	MEMSET(ADR(stMetsEfficiency.PackProduced), 16#00, SIZEOF(stMetsEfficiency.PackProduced));
	MEMSET(ADR(stMetsEfficiency.OutersProduced), 16#00, SIZEOF(stMetsEfficiency.OutersProduced));
	MEMSET(ADR(stMetsEfficiency.CaseProduced), 16#00, SIZEOF(stMetsEfficiency.CaseProduced));

	stMetsEfficiency.MachineID.ProductionSite	 := sProductionSite;
	stMetsEfficiency.MachineID.ProductionLine	:= sPCM;
	stMetsEfficiency.StartDateTime 			:= F_SYSTEM_SystemTimeAsISO8601(stCTDateTime.sSystemTime, stCTDateTime.sUTCTimeZoneOffset );
	stMetsEfficiency.CodingAndTrackingMode 	:= stPCMStatus.nOpMode;
	stMetsEfficiency.AcceptanceLevel  			:= stPCMStatus.nAcceptanceLevel;
	stMetsEfficiency.PacksPerOuter			:= stPCMStatus.nPacksPerOuter;

	MEMSET(ADR(stBarGraph), 16#00, SIZEOF(stBarGraph));

	bTimerFlag:=TRUE;
END_IF

tofDoneTimer(IN:=bTimerFlag,PT:=t#5s, Q=>bDone);

END_FUNCTION_BLOCK

// ---- POUs/METS/Common LIB/06_KPI LIB/ClearStatistic/FB_KPI_ClearGeneraStatistic.TcPOU
FUNCTION_BLOCK FB_KPI_ClearGeneraStatistic
VAR_INPUT
	bExecute				: BOOL;
	stCTDateTime			: ST_SYSTEM_DateTime;	(* CaseTrace date/time structure *)
	sProductionSite		: STRING(4);
	sPCM				: STRING(4);
	bForceNovReset		: BOOL;
END_VAR
VAR_IN_OUT

	stPCMStatus			: ST_PCM_Status;

	stMetsCameras			: ST_NOVRAM_METS_Cameras;
	stMetsEfficiency		: ST_NOVRAM_METS_Inspection;
	stCasePackerSignals		: ST_NOVRAM_METS_DualInputs;
	stCaseInspactionLog		: ST_NOVRAM_METS_CaseInspactionLog;
	
	stShiftStatistic		: ST_NOVRAM_METS_EventCounters; 
	stProdStatistic			: ST_NOVRAM_METS_EventCounters; 

	stBarGraph			: ST_HMI_BarGraph;

	stWriteOACFileStatistic		: ST_FILE_WriteFileStatistic;	(*Move to METSEfficency one day*)
	stWriteCHMFileStatistic		: ST_FILE_WriteFileStatistic;	(*Move to METSEfficency one day*)

END_VAR
VAR_OUTPUT
	bDone				: BOOL;
END_VAR
VAR
	fbExecute 			: R_TRIG;
	bTimerFlag			: BOOL;
	tofDoneTimer			: TOF;

	nCounter				: INT;


END_VAR

(* rising edge of bExecute *)
fbExecute(CLK:= bExecute);

bTimerFlag:=FALSE;

IF fbExecute.Q THEN

	nCounter := nCounter +1;

	MEMSET(ADR(stMetsCameras), 16#00, SIZEOF(stMetsCameras));
	MEMSET(ADR(stMetsEfficiency), 16#00, SIZEOF(stMetsEfficiency));
	MEMSET(ADR(stCasePackerSignals), 16#00, SIZEOF(stCasePackerSignals));
	MEMSET(ADR(stCaseInspactionLog), 16#00, SIZEOF(stCaseInspactionLog));

	stMetsCameras.MachineID.ProductionSite 	:= sProductionSite;
	stMetsCameras.MachineID.ProductionLine	:= sPCM;
	stMetsCameras.StartDateTime 				:=  F_SYSTEM_SystemTimeAsISO8601(stCTDateTime.sSystemTime, stCTDateTime.sUTCTimeZoneOffset );
	stMetsCameras.CodingAndTrackingMode 	:= stPCMStatus.nOpMode;

	stMetsEfficiency.MachineID.ProductionSite	 := sProductionSite;
	stMetsEfficiency.MachineID.ProductionLine	:= sPCM;
	stMetsEfficiency.StartDateTime 			:= F_SYSTEM_SystemTimeAsISO8601(stCTDateTime.sSystemTime, stCTDateTime.sUTCTimeZoneOffset );
	stMetsEfficiency.CodingAndTrackingMode 	:= stPCMStatus.nOpMode;
	stMetsEfficiency.AcceptanceLevel  			:= stPCMStatus.nAcceptanceLevel;
	stMetsEfficiency.PacksPerOuter			:= stPCMStatus.nPacksPerOuter;

	stCasePackerSignals.MachineID.ProductionSite	 := sProductionSite;
	stCasePackerSignals.MachineID.ProductionLine	:= sPCM;
	stCasePackerSignals.StartDateTime 				:=  F_SYSTEM_SystemTimeAsISO8601(stCTDateTime.sSystemTime, stCTDateTime.sUTCTimeZoneOffset );
	stCasePackerSignals.CodingAndTrackingMode	 	:=stPCMStatus.nOpMode;

	stCaseInspactionLog.MachineID.ProductionSite 	:= sProductionSite;
	stCaseInspactionLog.MachineID.ProductionLine	:= sPCM;
	stCaseInspactionLog.StartDateTime 				:=  F_SYSTEM_SystemTimeAsISO8601(stCTDateTime.sSystemTime, stCTDateTime.sUTCTimeZoneOffset );
	stCaseInspactionLog.CodingAndTrackingMode		:= stPCMStatus.nOpMode;
	stCaseInspactionLog.nPacksPerCase  			:= stPCMStatus.nPacksPerCase;
	stCaseInspactionLog.nOutersPerCase			:= stPCMStatus.nOutersPerCase;

	MEMSET(ADR(stBarGraph), 16#00, SIZEOF(stBarGraph));

	MEMSET(ADR(stWriteOACFileStatistic), 16#00, SIZEOF(stWriteOACFileStatistic));
	MEMSET(ADR(stWriteCHMFileStatistic), 16#00, SIZEOF(stWriteCHMFileStatistic));

	bTimerFlag:=TRUE;
END_IF

tofDoneTimer(IN:=bTimerFlag,PT:=t#5s, Q=>bDone);

IF bForceNovReset THEN
	MEMSET(ADR(stShiftStatistic), 16#00, SIZEOF(stShiftStatistic));
	MEMSET(ADR(stProdStatistic), 16#00, SIZEOF(stProdStatistic));
END_IF

END_FUNCTION_BLOCK

// ---- POUs/METS/Common LIB/06_KPI LIB/ClearStatistic/FB_KPI_ClearInspectionStatistic.TcPOU
FUNCTION_BLOCK FB_KPI_ClearInspectionStatistic
VAR_INPUT
	bExecute						: BOOL;
	stCTDateTime					: ST_SYSTEM_DateTime;	(* CaseTrace date/time structure *)
	nLowerCameraGroupIndex		: INT;
	nUpperCameraGroupIndex		: INT;
END_VAR
VAR_IN_OUT
	stEfficiencyToBeCleared			: ST_KPI_InspectionEfficency;
	stMetsCameras					: ST_NOVRAM_METS_Cameras;
END_VAR
VAR_OUTPUT
	bDone				: BOOL;
END_VAR
VAR
	fbExecute 			: R_TRIG;
	bTimerFlag			: BOOL;
	tofDoneTimer			: TOF;
	nIndex				: INT;

	nCounter				: INT;
END_VAR

(* rising edge of bExecute *)
fbExecute(CLK:= bExecute);

bTimerFlag:=FALSE;

IF fbExecute.Q THEN

	nCounter := nCounter +1;



	MEMSET(ADR(stEfficiencyToBeCleared), 16#00, SIZEOF(stEfficiencyToBeCleared));

	(*stEfficiencyToBeCleared.StartDateTime 			:= F_SYSTEM_SystemTimeAsISO8601(stCTDateTime.sSystemTime, stCTDateTime.sUTCTimeZoneOffset );*)

	IF nLowerCameraGroupIndex > 0 	AND
		nLowerCameraGroupIndex <= nUpperCameraGroupIndex THEN

		FOR nIndex :=nLowerCameraGroupIndex  TO MIN(nUpperCameraGroupIndex, cMAX_CAMERA_NUMBER)  DO
			MEMSET(ADR(stMetsCameras.aCameraEvaluation[nIndex]), 16#00, SIZEOF(stMetsCameras.aCameraEvaluation[nIndex]));
		END_FOR
	END_IF

	bTimerFlag:=TRUE;
END_IF

tofDoneTimer(IN:=bTimerFlag,PT:=t#5s, Q=>bDone);

END_FUNCTION_BLOCK

// ---- POUs/METS/Common LIB/06_KPI LIB/ClearStatistic/FB_KPI_ClearPackOuterInspection.TcPOU
FUNCTION_BLOCK FB_KPI_ClearPackOuterInspection
VAR_INPUT
	bExecute						: BOOL;
	stCTDateTime					: ST_SYSTEM_DateTime;	(* CaseTrace date/time structure *)
	sProductionSite				: STRING(4);
	sPCM						: STRING(4);
END_VAR
VAR_IN_OUT

	stPCMStatus					: ST_PCM_Status;
	stMetsEfficiency		: ST_NOVRAM_METS_Inspection;

END_VAR
VAR_OUTPUT
	bDone				: BOOL;
END_VAR
VAR
	fbExecute 			: R_TRIG;
	bTimerFlag			: BOOL;
	tofDoneTimer			: TOF;

	nCounter				: INT;
END_VAR

(* rising edge of bExecute *)
fbExecute(CLK:= bExecute);

bTimerFlag:=FALSE;

IF fbExecute.Q THEN

	nCounter := nCounter +1;

	stMetsEfficiency.MachineID.ProductionSite	 := sProductionSite;
	stMetsEfficiency.MachineID.ProductionLine	:= sPCM;
	stMetsEfficiency.StartDateTime 			:= F_SYSTEM_SystemTimeAsISO8601(stCTDateTime.sSystemTime, stCTDateTime.sUTCTimeZoneOffset );
	stMetsEfficiency.CodingAndTrackingMode 	:= stPCMStatus.nOpMode;
	stMetsEfficiency.AcceptanceLevel  			:= stPCMStatus.nAcceptanceLevel;
	stMetsEfficiency.PacksPerOuter			:= stPCMStatus.nPacksPerOuter;

	MEMSET(ADR(stMetsEfficiency.OutersProcessing), 16#00, SIZEOF(stMetsEfficiency.OutersProcessing));
	MEMSET(ADR(stMetsEfficiency.OCVFileEfficiency), 16#00, SIZEOF(stMetsEfficiency.OCVFileEfficiency));
	MEMSET(ADR(stMetsEfficiency.PacksRead), 16#00, SIZEOF(stMetsEfficiency.PacksRead));
	MEMSET(ADR(stMetsEfficiency.PackPosEfficiency), 16#00, SIZEOF(stMetsEfficiency.PackPosEfficiency));

	MEMSET(ADR(stMetsEfficiency.PackAggregationEfficiency), 16#00, SIZEOF(stMetsEfficiency.PackAggregationEfficiency));

	MEMSET(ADR(stMetsEfficiency.aConfirmCodeEfficiency), 16#00, SIZEOF(stMetsEfficiency.aConfirmCodeEfficiency));
	MEMSET(ADR(stMetsEfficiency.PackConfirmationEfficiency), 16#00, SIZEOF(stMetsEfficiency.PackConfirmationEfficiency));
	MEMSET(ADR(stMetsEfficiency.OuterValidationEfficiency), 16#00, SIZEOF(stMetsEfficiency.OuterValidationEfficiency));
	MEMSET(ADR(stMetsEfficiency.OuterAggregationEfficiency), 16#00, SIZEOF(stMetsEfficiency.OuterAggregationEfficiency));

	bTimerFlag:=TRUE;
END_IF

tofDoneTimer(IN:=bTimerFlag,PT:=t#5s, Q=>bDone);

END_FUNCTION_BLOCK

// ---- POUs/METS/Common LIB/06_KPI LIB/ItemEfficiency/FB_KPI_CaseEfficiency.TcPOU
FUNCTION_BLOCK FB_KPI_CaseEfficiency
VAR_INPUT
	bUpdateItemData		: 	BOOL;
	bItemSuccessful		:	 BOOL;
END_VAR
VAR_IN_OUT
	stItemInspection		: 	ST_KPI_InspectionEfficency;
END_VAR
VAR_OUTPUT
END_VAR
VAR
	rtrigUpdateItemData	:	 R_TRIG;
END_VAR

rtrigUpdateItemData(CLK:= bUpdateItemData);

IF rtrigUpdateItemData.Q THEN

	stItemInspection.ProcessedTotal :=  stItemInspection.ProcessedTotal + 1;
		IF bItemSuccessful THEN
			stItemInspection.ProcessedSuccessful := stItemInspection.ProcessedSuccessful + 1;
		ELSE
			stItemInspection.ProcessedRejected := stItemInspection.ProcessedRejected + 1;
		END_IF
END_IF

stItemInspection.ProcessedEfficiency := F_SafeDIV(stItemInspection.ProcessedSuccessful  * 100,  stItemInspection.ProcessedTotal);
stItemInspection.ProcessedEfficiency :=LIMIT(0, stItemInspection.ProcessedEfficiency, 100);

END_FUNCTION_BLOCK

// ---- POUs/METS/Common LIB/06_KPI LIB/ItemEfficiency/FB_KPI_InterimEfficiency.TcPOU
FUNCTION_BLOCK FB_KPI_InterimEfficiency
VAR_INPUT
	bUpdateItemData		: 	BOOL;
	bItemSuccessful		:	 BOOL;
END_VAR
VAR_IN_OUT
	stItemInspection		: 	ST_KPI_InspectionEfficency;
END_VAR
VAR_OUTPUT
END_VAR
VAR
	rtrigUpdateItemData	:	 R_TRIG;
END_VAR

rtrigUpdateItemData(CLK:= bUpdateItemData);

IF rtrigUpdateItemData.Q THEN

	stItemInspection.ProcessedTotal :=  stItemInspection.ProcessedTotal + 1;
		IF bItemSuccessful THEN
			stItemInspection.ProcessedSuccessful := stItemInspection.ProcessedSuccessful + 1;
		ELSE
			stItemInspection.ProcessedRejected := stItemInspection.ProcessedRejected + 1;
		END_IF
END_IF

stItemInspection.ProcessedEfficiency := F_SafeDIV(stItemInspection.ProcessedSuccessful  * 100,  stItemInspection.ProcessedTotal);
stItemInspection.ProcessedEfficiency :=LIMIT(0, stItemInspection.ProcessedEfficiency, 100);

END_FUNCTION_BLOCK

// ---- POUs/METS/Common LIB/06_KPI LIB/ItemEfficiency/FB_KPI_OutersEfficiency.TcPOU
FUNCTION_BLOCK FB_KPI_OutersEfficiency
VAR_INPUT
	ePackAggregationMode			: E_SYSTEM_PackAggregationMode ;
	bUpdateAtConfimrationCamera	: BOOL;
	bUpdateAtValidationCamera		: BOOL;
	bUpdateTotal						: BOOL;
	bUpdateConfirmCam				: BOOL;
	bUpdateValidCam					: BOOL;

	bItemSuccessful					: BOOL;

	nPackEntireLength					: INT;
	nOuterEntireLength				: INT;
	nValidCamExpectedResp			: INT;

END_VAR
VAR_IN_OUT
	stConfirmationCameraImage		: ST_SCANNER_ImageData;		(* image data structure *)
	stValidationCameraImage			: ST_SCANNER_ImageData;		(* image data structure *)

	stMetsEfficiency					: ST_NOVRAM_METS_Inspection;
END_VAR
VAR_OUTPUT
END_VAR
VAR
	rtrigUpdateAtConfimrationCamera	: R_TRIG;
	rtrigUpdateAtValidationCamera	: R_TRIG;
	rtrigUpdateTotal				: R_TRIG;
	rtrigUpdateConfirmCamera		: R_TRIG;
	rtrigUpdateValidCamera			: R_TRIG;
	rtrigUpdateKPI					: R_TRIG;

	nCodeLoopPerPos				: INT;

END_VAR

CASE ePackAggregationMode OF

	E_SYSTEM_PAOL_2CAM:

		SFLX();

	E_SYSTEM_PAOL_3CAM:

		PAOL();

	E_SYSTEM_PLAS_T01, E_SYSTEM_PLAS_T02, E_SYSTEM_PLAS_T03, E_SYSTEM_PLAS_T04:

		PLAS();

END_CASE

ACTION NCW:
rtrigUpdateTotal(CLK:= bUpdateTotal);

IF rtrigUpdateTotal.Q THEN

	stMetsEfficiency.OuterAggregationEfficiency.ProcessedTotal :=  stMetsEfficiency.OuterAggregationEfficiency.ProcessedTotal + 1;
		IF bItemSuccessful THEN
			stMetsEfficiency.OuterAggregationEfficiency.ProcessedSuccessful := stMetsEfficiency.OuterAggregationEfficiency.ProcessedSuccessful + 1;
		ELSE
			stMetsEfficiency.OuterAggregationEfficiency.ProcessedRejected := stMetsEfficiency.OuterAggregationEfficiency.ProcessedRejected + 1;
		END_IF
END_IF

stMetsEfficiency.OuterAggregationEfficiency.ProcessedEfficiency :=  F_SafeDIV( UDINT_TO_LREAL(stMetsEfficiency.OuterAggregationEfficiency.ProcessedSuccessful),
																	UDINT_TO_LREAL(stMetsEfficiency.OuterAggregationEfficiency.ProcessedTotal))* 100.0;
stMetsEfficiency.OuterAggregationEfficiency.ProcessedEfficiency	:= LIMIT(0,stMetsEfficiency.OuterAggregationEfficiency.ProcessedEfficiency , 100);
END_ACTION

ACTION PAOL:
rtrigUpdateAtConfimrationCamera(CLK:= bUpdateAtConfimrationCamera);
rtrigUpdateAtValidationCamera(CLK:=bUpdateAtValidationCamera);
rtrigUpdateTotal(CLK:= bUpdateTotal);
rtrigUpdateConfirmCamera(CLK:=bUpdateConfirmCam);
rtrigUpdateValidCamera(CLK:=bUpdateValidCam);

IF rtrigUpdateAtConfimrationCamera.Q THEN
	stMetsEfficiency.OutersProcessing.AtConfimrationCamera := stMetsEfficiency.OutersProcessing.AtConfimrationCamera + 1;
END_IF

IF rtrigUpdateAtValidationCamera.Q THEN
	stMetsEfficiency.OutersProcessing.AtValidationCamera := stMetsEfficiency.OutersProcessing.AtValidationCamera + 1;
END_IF

IF rtrigUpdateTotal.Q THEN

	stMetsEfficiency.OuterAggregationEfficiency.ProcessedTotal :=stMetsEfficiency. OuterAggregationEfficiency.ProcessedTotal +1;

		IF bItemSuccessful THEN
			stMetsEfficiency.OuterAggregationEfficiency.ProcessedSuccessful := stMetsEfficiency.OuterAggregationEfficiency.ProcessedSuccessful +1;
		ELSE
			stMetsEfficiency.OuterAggregationEfficiency.ProcessedRejected  := stMetsEfficiency.OuterAggregationEfficiency.ProcessedRejected +1;
		END_IF

	stMetsEfficiency.OuterAggregationEfficiency.ProcessedEfficiency :=  F_SafeDIV( UDINT_TO_LREAL(stMetsEfficiency.OuterAggregationEfficiency.ProcessedSuccessful),
																		UDINT_TO_LREAL(stMetsEfficiency.OuterAggregationEfficiency.ProcessedTotal))* 100.0;
	stMetsEfficiency.OuterAggregationEfficiency.ProcessedEfficiency	:= LIMIT(0,stMetsEfficiency.OuterAggregationEfficiency.ProcessedEfficiency , 100);
END_IF

(************************* Update Pack Confirmation Process Efficiency*******************************************************************************)

IF rtrigUpdateConfirmCamera.Q  THEN

	stMetsEfficiency.PackConfirmationEfficiency.ProcessedTotal	:= 	stMetsEfficiency.PackConfirmationEfficiency.ProcessedTotal +1;

	IF F_PACK_ValidateCodeASCII(stConfirmationCameraImage.aCodeData[1].strDataString) =  nPackEntireLength			OR
			F_PACK_ValidateCodeASCII(stConfirmationCameraImage.aCodeData[2].strDataString) =  nPackEntireLength 	THEN

		stMetsEfficiency.PackConfirmationEfficiency.ProcessedSuccessful :=  stMetsEfficiency.PackConfirmationEfficiency.ProcessedSuccessful +1;
	ELSE
		stMetsEfficiency.PackConfirmationEfficiency.ProcessedRejected :=  stMetsEfficiency.PackConfirmationEfficiency.ProcessedRejected +1;
	END_IF

(*Confirmation Cameras Individual per pack*)
	FOR nCodeLoopPerPos := 1 TO 2 DO
		CASE LREAL_TO_INT(stConfirmationCameraImage.aCodeData[nCodeLoopPerPos].nProgramNo) OF
			1:
				IF F_PACK_ValidateCodeASCII(stConfirmationCameraImage.aCodeData[nCodeLoopPerPos].strDataString) =  nPackEntireLength THEN
					stMetsEfficiency.aConfirmCodeEfficiency[1].ReadOK :=  stMetsEfficiency.aConfirmCodeEfficiency[1].ReadOK +1;
				END_IF
			2:
				IF F_PACK_ValidateCodeASCII(stConfirmationCameraImage.aCodeData[nCodeLoopPerPos].strDataString) =  nPackEntireLength THEN
					stMetsEfficiency.aConfirmCodeEfficiency[2].ReadOK := stMetsEfficiency. aConfirmCodeEfficiency[2].ReadOK +1;
				END_IF
		END_CASE
	END_FOR

	stMetsEfficiency.PackConfirmationEfficiency.ProcessedEfficiency :=  F_SafeDIV( UDINT_TO_LREAL(stMetsEfficiency.PackConfirmationEfficiency.ProcessedSuccessful),
																	UDINT_TO_LREAL(stMetsEfficiency.PackConfirmationEfficiency.ProcessedTotal))* 100.0;
	stMetsEfficiency.PackConfirmationEfficiency.ProcessedEfficiency	:= LIMIT(0,stMetsEfficiency.PackConfirmationEfficiency.ProcessedEfficiency, 100);

	stMetsEfficiency.aConfirmCodeEfficiency[1].Efficiency :=  F_SafeDIV( UDINT_TO_LREAL(stMetsEfficiency.aConfirmCodeEfficiency[1].ReadOK),
																	UDINT_TO_LREAL(stMetsEfficiency.PackConfirmationEfficiency.ProcessedTotal))* 100.0;
	stMetsEfficiency.aConfirmCodeEfficiency[1].Efficiency	:= LIMIT(0,stMetsEfficiency.aConfirmCodeEfficiency[1].Efficiency, 100);

	stMetsEfficiency.aConfirmCodeEfficiency[2].Efficiency :=  F_SafeDIV( UDINT_TO_LREAL(stMetsEfficiency.aConfirmCodeEfficiency[2].ReadOK),
																	UDINT_TO_LREAL(stMetsEfficiency.PackConfirmationEfficiency.ProcessedTotal))* 100.0;
	stMetsEfficiency.aConfirmCodeEfficiency[2].Efficiency	:= LIMIT(0,stMetsEfficiency.aConfirmCodeEfficiency[2].Efficiency , 100);

END_IF

(************************* Update Outer Validation Process Efficiency*******************************************************************************)

IF rtrigUpdateValidCamera.Q  THEN

	stMetsEfficiency.OuterValidationEfficiency.ProcessedTotal :=	stMetsEfficiency.OuterValidationEfficiency.ProcessedTotal + 1;

	IF LEN(stValidationCameraImage.aCodeData[1].strDataString) =  nOuterEntireLength 				OR
		LEN(stValidationCameraImage.aCodeData[2].strDataString) =  nOuterEntireLength 				THEN

		stMetsEfficiency.OuterValidationEfficiency.ProcessedSuccessful :=  stMetsEfficiency.OuterValidationEfficiency.ProcessedSuccessful +1;
	END_IF

(*Vaidation Cameras Individual read*)
	IF nValidCamExpectedResp = 2 THEN
		FOR nCodeLoopPerPos := 1 TO 2 DO
			CASE LREAL_TO_INT(stValidationCameraImage.aCodeData[nCodeLoopPerPos].nProgramNo) OF
				1:
					IF LEN(stValidationCameraImage.aCodeData[nCodeLoopPerPos].strDataString) =  nOuterEntireLength THEN
						stMetsEfficiency.aValidCodeEfficiency[1].ReadOK :=  stMetsEfficiency.aValidCodeEfficiency[1].ReadOK +1;
					END_IF
				2:
					IF LEN(stValidationCameraImage.aCodeData[nCodeLoopPerPos].strDataString) =  nOuterEntireLength THEN
						stMetsEfficiency.aValidCodeEfficiency[2].ReadOK := stMetsEfficiency. aValidCodeEfficiency[2].ReadOK +1;
					END_IF
			END_CASE
		END_FOR
	ELSIF nValidCamExpectedResp = 1 THEN
		IF LEN(stValidationCameraImage.aCodeData[1].strDataString) =  nOuterEntireLength THEN
			stMetsEfficiency.aValidCodeEfficiency[1].ReadOK :=  stMetsEfficiency.aValidCodeEfficiency[1].ReadOK +1;
		END_IF
	END_IF


	stMetsEfficiency.OuterValidationEfficiency.ProcessedEfficiency :=  F_SafeDIV( UDINT_TO_LREAL(stMetsEfficiency.OuterValidationEfficiency.ProcessedSuccessful),
																		UDINT_TO_LREAL(stMetsEfficiency.OuterValidationEfficiency.ProcessedTotal))* 100.0;
	stMetsEfficiency.OuterValidationEfficiency.ProcessedEfficiency	:= LIMIT(0,stMetsEfficiency.OuterValidationEfficiency.ProcessedEfficiency, 100);

	stMetsEfficiency.aValidCodeEfficiency[1].Efficiency :=  F_SafeDIV( UDINT_TO_LREAL(stMetsEfficiency.aValidCodeEfficiency[1].ReadOK),
																	UDINT_TO_LREAL(stMetsEfficiency.OuterValidationEfficiency.ProcessedTotal))* 100.0;
	stMetsEfficiency.aValidCodeEfficiency[1].Efficiency	:= LIMIT(0,stMetsEfficiency.aValidCodeEfficiency[1].Efficiency, 100);

	stMetsEfficiency.aValidCodeEfficiency[2].Efficiency :=  F_SafeDIV( UDINT_TO_LREAL(stMetsEfficiency.aValidCodeEfficiency[2].ReadOK),
																	UDINT_TO_LREAL(stMetsEfficiency.OuterValidationEfficiency.ProcessedTotal))* 100.0;
	stMetsEfficiency.aValidCodeEfficiency[2].Efficiency	:= LIMIT(0,stMetsEfficiency.aValidCodeEfficiency[2].Efficiency , 100);

END_IF
END_ACTION

ACTION PLAS:
rtrigUpdateAtConfimrationCamera(CLK:= bUpdateAtConfimrationCamera);
rtrigUpdateAtValidationCamera(CLK:=bUpdateAtValidationCamera);
rtrigUpdateTotal(CLK:= bUpdateTotal);
rtrigUpdateConfirmCamera(CLK:=bUpdateConfirmCam);
rtrigUpdateValidCamera(CLK:=bUpdateValidCam);

IF rtrigUpdateAtConfimrationCamera.Q THEN
	stMetsEfficiency.OutersProcessing.AtConfimrationCamera := stMetsEfficiency.OutersProcessing.AtConfimrationCamera + 1;
END_IF

IF rtrigUpdateAtValidationCamera.Q THEN
	stMetsEfficiency.OutersProcessing.AtValidationCamera := stMetsEfficiency.OutersProcessing.AtValidationCamera + 1;
END_IF

IF rtrigUpdateTotal.Q THEN

	stMetsEfficiency.OuterAggregationEfficiency.ProcessedTotal :=stMetsEfficiency. OuterAggregationEfficiency.ProcessedTotal +1;

		IF bItemSuccessful THEN
			stMetsEfficiency.OuterAggregationEfficiency.ProcessedSuccessful := stMetsEfficiency.OuterAggregationEfficiency.ProcessedSuccessful +1;
		ELSE
			stMetsEfficiency.OuterAggregationEfficiency.ProcessedRejected  := stMetsEfficiency.OuterAggregationEfficiency.ProcessedRejected +1;
		END_IF

	stMetsEfficiency.OuterAggregationEfficiency.ProcessedEfficiency :=  F_SafeDIV( UDINT_TO_LREAL(stMetsEfficiency.OuterAggregationEfficiency.ProcessedSuccessful),
																		UDINT_TO_LREAL(stMetsEfficiency.OuterAggregationEfficiency.ProcessedTotal))* 100.0;
	stMetsEfficiency.OuterAggregationEfficiency.ProcessedEfficiency	:= LIMIT(0,stMetsEfficiency.OuterAggregationEfficiency.ProcessedEfficiency , 100);
END_IF

(************************* Update Pack Confirmation Process Efficiency*******************************************************************************)

IF rtrigUpdateConfirmCamera.Q  THEN

	stMetsEfficiency.PackConfirmationEfficiency.ProcessedTotal	:= 	stMetsEfficiency.PackConfirmationEfficiency.ProcessedTotal +1;

	IF F_PACK_ValidateCodeASCII(stConfirmationCameraImage.aCodeData[1].strDataString) =  nPackEntireLength			OR
			F_PACK_ValidateCodeASCII(stConfirmationCameraImage.aCodeData[2].strDataString) =  nPackEntireLength 	THEN

		stMetsEfficiency.PackConfirmationEfficiency.ProcessedSuccessful :=  stMetsEfficiency.PackConfirmationEfficiency.ProcessedSuccessful +1;
	ELSE
		stMetsEfficiency.PackConfirmationEfficiency.ProcessedRejected :=  stMetsEfficiency.PackConfirmationEfficiency.ProcessedRejected +1;
	END_IF

(*Confirmation Cameras Individual per pack*)
	FOR nCodeLoopPerPos := 1 TO 2 DO
		CASE LREAL_TO_INT(stConfirmationCameraImage.aCodeData[nCodeLoopPerPos].nProgramNo) OF
			1:
				IF F_PACK_ValidateCodeASCII(stConfirmationCameraImage.aCodeData[nCodeLoopPerPos].strDataString) =  nPackEntireLength THEN
					stMetsEfficiency.aConfirmCodeEfficiency[1].ReadOK :=  stMetsEfficiency.aConfirmCodeEfficiency[1].ReadOK +1;
				END_IF
			2:
				IF F_PACK_ValidateCodeASCII(stConfirmationCameraImage.aCodeData[nCodeLoopPerPos].strDataString) =  nPackEntireLength THEN
					stMetsEfficiency.aConfirmCodeEfficiency[2].ReadOK := stMetsEfficiency. aConfirmCodeEfficiency[2].ReadOK +1;
				END_IF
		END_CASE
	END_FOR

	stMetsEfficiency.PackConfirmationEfficiency.ProcessedEfficiency :=  F_SafeDIV( UDINT_TO_LREAL(stMetsEfficiency.PackConfirmationEfficiency.ProcessedSuccessful),
																	UDINT_TO_LREAL(stMetsEfficiency.PackConfirmationEfficiency.ProcessedTotal))* 100.0;
	stMetsEfficiency.PackConfirmationEfficiency.ProcessedEfficiency	:= LIMIT(0,stMetsEfficiency.PackConfirmationEfficiency.ProcessedEfficiency, 100);

	stMetsEfficiency.aConfirmCodeEfficiency[1].Efficiency :=  F_SafeDIV( UDINT_TO_LREAL(stMetsEfficiency.aConfirmCodeEfficiency[1].ReadOK),
																	UDINT_TO_LREAL(stMetsEfficiency.PackConfirmationEfficiency.ProcessedTotal))* 100.0;
	stMetsEfficiency.aConfirmCodeEfficiency[1].Efficiency	:= LIMIT(0,stMetsEfficiency.aConfirmCodeEfficiency[1].Efficiency, 100);

	stMetsEfficiency.aConfirmCodeEfficiency[2].Efficiency :=  F_SafeDIV( UDINT_TO_LREAL(stMetsEfficiency.aConfirmCodeEfficiency[2].ReadOK),
																	UDINT_TO_LREAL(stMetsEfficiency.PackConfirmationEfficiency.ProcessedTotal))* 100.0;
	stMetsEfficiency.aConfirmCodeEfficiency[2].Efficiency	:= LIMIT(0,stMetsEfficiency.aConfirmCodeEfficiency[2].Efficiency , 100);

END_IF

(************************* Update Outer Validation Process Efficiency*******************************************************************************)

IF rtrigUpdateValidCamera.Q  THEN

	stMetsEfficiency.OuterValidationEfficiency.ProcessedTotal :=	stMetsEfficiency.OuterValidationEfficiency.ProcessedTotal + 1;

	IF LEN(stValidationCameraImage.aCodeData[1].strDataString) =  nOuterEntireLength 				OR
		LEN(stValidationCameraImage.aCodeData[2].strDataString) =  nOuterEntireLength 				THEN

		stMetsEfficiency.OuterValidationEfficiency.ProcessedSuccessful :=  stMetsEfficiency.OuterValidationEfficiency.ProcessedSuccessful +1;
	END_IF

(*Vaidation Cameras Individual read*)
	IF nValidCamExpectedResp = 2 THEN
		FOR nCodeLoopPerPos := 1 TO 2 DO
			CASE LREAL_TO_INT(stValidationCameraImage.aCodeData[nCodeLoopPerPos].nProgramNo) OF
				1:
					IF LEN(stValidationCameraImage.aCodeData[nCodeLoopPerPos].strDataString) =  nOuterEntireLength THEN
						stMetsEfficiency.aValidCodeEfficiency[1].ReadOK :=  stMetsEfficiency.aValidCodeEfficiency[1].ReadOK +1;
					END_IF
				2:
					IF LEN(stValidationCameraImage.aCodeData[nCodeLoopPerPos].strDataString) =  nOuterEntireLength THEN
						stMetsEfficiency.aValidCodeEfficiency[2].ReadOK := stMetsEfficiency. aValidCodeEfficiency[2].ReadOK +1;
					END_IF
			END_CASE
		END_FOR
	ELSIF nValidCamExpectedResp = 1 THEN
		IF LEN(stValidationCameraImage.aCodeData[1].strDataString) =  nOuterEntireLength THEN
			stMetsEfficiency.aValidCodeEfficiency[1].ReadOK :=  stMetsEfficiency.aValidCodeEfficiency[1].ReadOK +1;
		END_IF
	END_IF

	stMetsEfficiency.OuterValidationEfficiency.ProcessedEfficiency :=  F_SafeDIV( UDINT_TO_LREAL(stMetsEfficiency.OuterValidationEfficiency.ProcessedSuccessful),
																		UDINT_TO_LREAL(stMetsEfficiency.OuterValidationEfficiency.ProcessedTotal))* 100.0;
	stMetsEfficiency.OuterValidationEfficiency.ProcessedEfficiency	:= LIMIT(0,stMetsEfficiency.OuterValidationEfficiency.ProcessedEfficiency, 100);

	stMetsEfficiency.aValidCodeEfficiency[1].Efficiency :=  F_SafeDIV( UDINT_TO_LREAL(stMetsEfficiency.aValidCodeEfficiency[1].ReadOK),
																	UDINT_TO_LREAL(stMetsEfficiency.OuterValidationEfficiency.ProcessedTotal))* 100.0;
	stMetsEfficiency.aValidCodeEfficiency[1].Efficiency	:= LIMIT(0,stMetsEfficiency.aValidCodeEfficiency[1].Efficiency, 100);

	stMetsEfficiency.aValidCodeEfficiency[2].Efficiency :=  F_SafeDIV( UDINT_TO_LREAL(stMetsEfficiency.aValidCodeEfficiency[2].ReadOK),
																	UDINT_TO_LREAL(stMetsEfficiency.OuterValidationEfficiency.ProcessedTotal))* 100.0;
	stMetsEfficiency.aValidCodeEfficiency[2].Efficiency	:= LIMIT(0,stMetsEfficiency.aValidCodeEfficiency[2].Efficiency , 100);

END_IF
END_ACTION

ACTION SFLX:

rtrigUpdateAtValidationCamera(CLK:=bUpdateAtValidationCamera);
rtrigUpdateTotal(CLK:= bUpdateTotal);
rtrigUpdateValidCamera(CLK:=bUpdateValidCam);

IF rtrigUpdateAtValidationCamera.Q THEN
	stMetsEfficiency.OutersProcessing.AtValidationCamera := stMetsEfficiency.OutersProcessing.AtValidationCamera + 1;
END_IF

IF rtrigUpdateTotal.Q THEN

	stMetsEfficiency.OuterAggregationEfficiency.ProcessedTotal :=stMetsEfficiency. OuterAggregationEfficiency.ProcessedTotal +1;

		IF bItemSuccessful THEN
			stMetsEfficiency.OuterAggregationEfficiency.ProcessedSuccessful := stMetsEfficiency.OuterAggregationEfficiency.ProcessedSuccessful +1;
		ELSE
			stMetsEfficiency.OuterAggregationEfficiency.ProcessedRejected  := stMetsEfficiency.OuterAggregationEfficiency.ProcessedRejected +1;
		END_IF

	stMetsEfficiency.OuterAggregationEfficiency.ProcessedEfficiency :=  F_SafeDIV( UDINT_TO_LREAL(stMetsEfficiency.OuterAggregationEfficiency.ProcessedSuccessful),
																		UDINT_TO_LREAL(stMetsEfficiency.OuterAggregationEfficiency.ProcessedTotal))* 100.0;
	stMetsEfficiency.OuterAggregationEfficiency.ProcessedEfficiency	:= LIMIT(0,stMetsEfficiency.OuterAggregationEfficiency.ProcessedEfficiency , 100);
END_IF

(************************* Update Outer Validation Process Efficiency*******************************************************************************)

IF rtrigUpdateValidCamera.Q  THEN

	stMetsEfficiency.OuterValidationEfficiency.ProcessedTotal :=	stMetsEfficiency.OuterValidationEfficiency.ProcessedTotal + 1;

	IF LEN(stValidationCameraImage.aCodeData[1].strDataString) =  nOuterEntireLength 				OR
		LEN(stValidationCameraImage.aCodeData[2].strDataString) =  nOuterEntireLength 				THEN

		stMetsEfficiency.OuterValidationEfficiency.ProcessedSuccessful :=  stMetsEfficiency.OuterValidationEfficiency.ProcessedSuccessful +1;
	END_IF

(*Vaidation Cameras Individual read*)

	IF LEN(stValidationCameraImage.aCodeData[1].strDataString) =  nOuterEntireLength THEN
		stMetsEfficiency.aValidCodeEfficiency[1].ReadOK :=  stMetsEfficiency.aValidCodeEfficiency[1].ReadOK +1;
	END_IF

	stMetsEfficiency.OuterValidationEfficiency.ProcessedEfficiency :=  F_SafeDIV( UDINT_TO_LREAL(stMetsEfficiency.OuterValidationEfficiency.ProcessedSuccessful),
																		UDINT_TO_LREAL(stMetsEfficiency.OuterValidationEfficiency.ProcessedTotal))* 100.0;
	stMetsEfficiency.OuterValidationEfficiency.ProcessedEfficiency	:= LIMIT(0,stMetsEfficiency.OuterValidationEfficiency.ProcessedEfficiency, 100);

	stMetsEfficiency.aValidCodeEfficiency[1].Efficiency :=  F_SafeDIV( UDINT_TO_LREAL(stMetsEfficiency.aValidCodeEfficiency[1].ReadOK),
																	UDINT_TO_LREAL(stMetsEfficiency.OuterValidationEfficiency.ProcessedTotal))* 100.0;
	stMetsEfficiency.aValidCodeEfficiency[1].Efficiency	:= LIMIT(0,stMetsEfficiency.aValidCodeEfficiency[1].Efficiency, 100);

END_IF
END_ACTION

END_FUNCTION_BLOCK

// ---- POUs/METS/Common LIB/06_KPI LIB/RejectCounters/FB_KPI_CaseLevelCounter.TcPOU
FUNCTION_BLOCK FB_KPI_CaseLevelCounter
VAR_INPUT
	bExecute					: BOOL;			(* set TRUE to add value to buffer *)
	stCTDateTime				: ST_SYSTEM_DateTime;	(* CaseTrace date/time structure *)
	nCaseRejectID				: UINT;
	aRejectCountersID			: ARRAY[0..cMAX_REJECT_REASON] OF UINT;
END_VAR
VAR_IN_OUT
	aShiftRejectCounters		: ARRAY[0..cMAX_REJECT_REASON] OF ST_LOG_RejectReasons;
	aProdRejectCounters		: ARRAY[0..cMAX_REJECT_REASON] OF ST_LOG_RejectReasons;
END_VAR
VAR_OUTPUT
	bDone					: BOOL;			(* TRUE = complete *)
END_VAR
VAR
	fbExecute					: R_TRIG;
	nMaxIndex				: UINT;

	nRejectIndex				: T_PositiveINT;

END_VAR

(* rising edge of bExecute *)
fbExecute(CLK:= bExecute);

(* search for strBarcode in queue *)
IF fbExecute.Q = TRUE THEN

	FOR nRejectIndex := 0  TO  cMAX_REJECT_REASON DO
		IF nCaseRejectID = aRejectCountersID[nRejectIndex] THEN

			aShiftRejectCounters[nRejectIndex].nRejectCounter := aShiftRejectCounters[nRejectIndex].nRejectCounter + 1;
			aShiftRejectCounters[nRejectIndex].stLastTimeStamp := stCTDateTime.sSystemTime;
		
			aProdRejectCounters[nRejectIndex].nRejectCounter := aProdRejectCounters[nRejectIndex].nRejectCounter + 1;
			aProdRejectCounters[nRejectIndex].stLastTimeStamp := stCTDateTime.sSystemTime;
			EXIT;
		END_IF
	END_FOR

	bDone := TRUE;

(* bExecute has been reset *)
ELSIF bExecute = FALSE THEN

	(* reset outputs *)
	bDone := FALSE;

END_IF

END_FUNCTION_BLOCK

// ---- POUs/METS/Common LIB/06_KPI LIB/RejectCounters/FB_KPI_OuterLevelCounter.TcPOU
FUNCTION_BLOCK FB_KPI_OuterLevelCounter
VAR_INPUT
	bExecute					: BOOL;			(* set TRUE to add value to buffer *)
	stCTDateTime				: ST_SYSTEM_DateTime;	(* CaseTrace date/time structure *)
	sOuterStatus				: ST_OUTER_Status;	(* Outer status *)
	aRejectCountersID			: ARRAY[0..cMAX_REJECT_REASON] OF UINT;
END_VAR
VAR_IN_OUT
	aShiftRejectCounters		: ARRAY[0..cMAX_REJECT_REASON] OF ST_LOG_RejectReasons;
	aProdRejectCounters		: ARRAY[0..cMAX_REJECT_REASON] OF ST_LOG_RejectReasons;
END_VAR
VAR_OUTPUT
	bDone					: BOOL;			(* TRUE = complete *)
END_VAR
VAR
	fbExecute					: R_TRIG;
	//nMaxIndex				: UINT;

	nRejectIndex				: T_PositiveINT;

END_VAR

(* rising edge of bExecute *)
fbExecute(CLK:= bExecute);

(* search for strBarcode in queue *)
IF fbExecute.Q = TRUE THEN

	FOR nRejectIndex := 0  TO  cMAX_REJECT_REASON DO
		IF sOuterStatus.stOACData.OuterRejectID = aRejectCountersID[nRejectIndex] THEN

			aShiftRejectCounters[nRejectIndex].nRejectCounter := aShiftRejectCounters[nRejectIndex].nRejectCounter + 1;
			aShiftRejectCounters[nRejectIndex].stLastTimeStamp := stCTDateTime.sSystemTime;

			aProdRejectCounters[nRejectIndex].nRejectCounter := aProdRejectCounters[nRejectIndex].nRejectCounter + 1;
			aProdRejectCounters[nRejectIndex].stLastTimeStamp := stCTDateTime.sSystemTime;
			EXIT;
		END_IF
	END_FOR

	bDone := TRUE;

(* bExecute has been reset *)
ELSIF bExecute = FALSE THEN

	(* reset outputs *)
	bDone := FALSE;

END_IF

END_FUNCTION_BLOCK

// ---- POUs/METS/Common LIB/06_KPI LIB/RejectCounters/FB_KPI_PackLevelCounter.TcPOU
FUNCTION_BLOCK FB_KPI_PackLevelCounter
VAR_INPUT
	bExecute					: BOOL;			(* set TRUE to add value to buffer *)
	stCTDateTime				: ST_SYSTEM_DateTime;	(* CaseTrace date/time structure *)
	stOuterStatus				: ST_OUTER_Status;	(* Outer status *)
	aRejectCountersID			: ARRAY[0..cMAX_REJECT_REASON] OF UINT;
END_VAR
VAR_IN_OUT
	aShiftRejectCounters		: ARRAY[0..cMAX_REJECT_REASON] OF ST_LOG_RejectReasons;
	aProdRejectCounters		: ARRAY[0..cMAX_REJECT_REASON] OF ST_LOG_RejectReasons;
END_VAR
VAR_OUTPUT
	bDone					: BOOL;			(* TRUE = complete *)
END_VAR
VAR
	fbExecute					: R_TRIG;
	//nMaxIndex				: UINT;
	nPackRejectChekIndex		: T_PositiveINT;
	nRejectIndex				: T_PositiveINT;

END_VAR

(* rising edge of bExecute *)
fbExecute(CLK:= bExecute);

(* search for strBarcode in queue *)
IF fbExecute.Q = TRUE THEN

	FOR nPackRejectChekIndex := 1 TO MIN(stOuterStatus.stOACData.NumberOfPacks, cMAX_PACKS_PER_OUTER) BY 1 DO
		FOR nRejectIndex := 0  TO  cMAX_REJECT_REASON DO
			IF stOuterStatus.stOACData.PackRejectID[nPackRejectChekIndex] = aRejectCountersID[nRejectIndex] THEN

				aShiftRejectCounters[nRejectIndex].nRejectCounter := aShiftRejectCounters[nRejectIndex].nRejectCounter + 1;
				aShiftRejectCounters[nRejectIndex].stLastTimeStamp := stCTDateTime.sSystemTime;

				aProdRejectCounters[nRejectIndex].nRejectCounter := aProdRejectCounters[nRejectIndex].nRejectCounter + 1;
				aProdRejectCounters[nRejectIndex].stLastTimeStamp := stCTDateTime.sSystemTime;
				EXIT;
			END_IF
		END_FOR
	END_FOR

	bDone := TRUE;

(* bExecute has been reset *)
ELSIF bExecute = FALSE THEN

	(* reset outputs *)
	bDone := FALSE;

END_IF

END_FUNCTION_BLOCK

// ---- POUs/METS/Common LIB/07_DEVICE LIB/Cylinders/FB_Cylinder.TcPOU
FUNCTION_BLOCK FB_Cylinder
VAR_INPUT

	bEnable				: BOOL;
	bManualMode			: BOOL;
	bAutoMode			: BOOL;

	eCylinderCommandAuto	: E_CYLINDER_Position := E_CYLINDER_Position.STOP;
	eCylinderCommandHMI	: E_CYLINDER_Position := E_CYLINDER_Position.STOP;
	tOperationTime		: TIME:=T#1S;
	tTimeOut				: TIME:=T#3S;

	bReleaseRetractPos		: BOOL;
	bReleaseExtendPos		: BOOL;

	bCylinderRetractedInput	: BOOL;
	bCylinderExtendedInput	: BOOL;

	bExtendAsHomePos 	: BOOL;
	sDeviceTagID			: STRING(10);
	sRetractTagID			: STRING(10);
	sExtendTagID			: STRING(10);

END_VAR
VAR_OUTPUT
	bDeviceDisable		: BOOL;
	bMoveNotAllowed		: BOOL;
	bErrorPosition			: BOOL;
	bInPosition			: BOOL;
	bHomePosition			: BOOL;
	bCylinderExtendOutput	: BOOL;
	bCylinderRetractOutput	: BOOL;
	bCylinderInRetractedPosition: BOOL;
	bCylinderInExtendedPosition: BOOL;
	bCylinderIsRetracting	: BOOL;
	bCylinderIsExtending	: BOOL;

	stTagID		:	ST_CYLINDER_TagID;

END_VAR
VAR
	ton_Retract	:	TON;
	ton_Extend	:	TON;
	ton_Timeout	:	TON;

	eCylinderCommand		: E_CYLINDER_Position := E_CYLINDER_Position.STOP;

END_VAR

stTagID.sDeviceTagID	:=	sDeviceTagID;
stTagID.sRetractTagID	:=	sRetractTagID;
stTagID.sExtendTagID	:=	sExtendTagID;

(********************************(Enable )**********************************************************)
IF NOT bEnable THEN

	bDeviceDisable		:=	TRUE;
	bMoveNotAllowed		:= 	TRUE;
	bErrorPosition			:=	FALSE;
	bInPosition			:=	TRUE;
	bHomePosition			:=	TRUE;
	bCylinderExtendOutput	:=	FALSE;
	bCylinderRetractOutput	:=	FALSE;
	bCylinderInRetractedPosition :=	FALSE;
	bCylinderInExtendedPosition :=	FALSE;
	bCylinderIsRetracting	:=	FALSE;
	bCylinderIsExtending	:=	FALSE;

	ton_Retract(IN := FALSE);
	ton_Extend(IN := FALSE);
	ton_Timeout(IN := FALSE);


	RETURN;
ELSE

	bDeviceDisable :=	FALSE;
END_IF

(********************************(Operational Mode )**********************************************************)

IF bManualMode THEN

	bMoveNotAllowed	:= FALSE;
	eCylinderCommand	:= eCylinderCommandHMI;
ELSIF bAutoMode THEN

	bMoveNotAllowed	:= FALSE;
	eCylinderCommand	:= eCylinderCommandAuto;
ELSE
	bMoveNotAllowed	:= TRUE;
END_IF
(********************************(Timers )**********************************************************)

(* E_CYLINDER_Position.EXTEND Timer **************************************)
IF	bCylinderExtendedInput	AND	NOT	bCylinderRetractedInput THEN

		ton_Extend.IN	:=	TRUE;
ELSE
		ton_Extend.IN	:=	FALSE;
END_IF

ton_Extend(IN:= , PT:= tOperationTime, Q=> bCylinderInExtendedPosition  , ET=> );

(* E_CYLINDER_Position.RETRACT Timer ***************************************)
IF 	bCylinderRetractedInput	AND	NOT	bCylinderExtendedInput THEN

		ton_Retract.IN	:=	TRUE;
ELSE
		ton_Retract.IN	:=	FALSE;
END_IF

ton_Retract(IN:= , PT:= tOperationTime, Q=> bCylinderInRetractedPosition  , ET=> );

(********************************(Home)**********************************************************)

bHomePosition		:=	 (bCylinderInRetractedPosition AND NOT bExtendAsHomePos)	OR
					(bCylinderInExtendedPosition AND bExtendAsHomePos);

(********************************( Sequence )*****************************************************)

CASE eCylinderCommand OF
E_CYLINDER_Position.EXTEND:

	bMoveNotAllowed	:= TRUE;

	IF bReleaseExtendPos THEN

		bCylinderExtendOutput					:=	TRUE;
		bCylinderRetractOutput					:= 	FALSE;

		IF   ton_Extend.Q THEN
			bInPosition						 := 	TRUE;
			bCylinderIsRetracting				:= 	FALSE;
			bCylinderIsExtending				:= 	FALSE;
		ELSE
			bInPosition						 :=  	FALSE;
			IF NOT ton_Retract.Q  THEN
				bCylinderIsRetracting				:= 	FALSE;
				bCylinderIsExtending				:= 	TRUE;
			END_IF
		END_IF

		bMoveNotAllowed	:= FALSE;
	END_IF

E_CYLINDER_Position.RETRACT:

	bMoveNotAllowed	:= TRUE;

	IF bReleaseRetractPos THEN

		bCylinderRetractOutput					:=	TRUE;
		bCylinderExtendOutput					:=	FALSE;

		IF   ton_Retract.Q THEN
			bInPosition						 := 	TRUE;
			bCylinderIsRetracting				:= 	FALSE;
			bCylinderIsExtending				:= 	FALSE;
		ELSE
			bInPosition						 :=  	FALSE;
			IF NOT ton_Extend.Q THEN
				bCylinderIsRetracting				:= 	TRUE;
				bCylinderIsExtending				:= 	FALSE;
			END_IF
		END_IF

		bMoveNotAllowed	:= FALSE;
	END_IF

E_CYLINDER_Position.STOP:

		IF NOT bReleaseRetractPos AND NOT bReleaseExtendPos THEN
			bMoveNotAllowed	:= TRUE;
		ELSE
			bMoveNotAllowed	:= FALSE;
		END_IF

		bCylinderExtendOutput					:=	FALSE;
		bCylinderRetractOutput					:=	FALSE;

		bInPosition							 :=   	TRUE;
		bCylinderIsRetracting					:= 	FALSE;
		bCylinderIsExtending					:= 	FALSE;
ELSE

		IF NOT bExtendAsHomePos THEN
			bCylinderExtendOutput					:=	FALSE;
			bCylinderRetractOutput					:=	TRUE;
		ELSE
			bCylinderExtendOutput					:=	TRUE;
			bCylinderRetractOutput					:=	FALSE;
		END_IF

		bInPosition							 :=   	FALSE;
		bCylinderIsRetracting					:= 	FALSE;
		bCylinderIsExtending					:= 	FALSE;
END_CASE


(*********************(Error Timer) **************************************)

IF	((bCylinderExtendOutput AND NOT bCylinderExtendedInput) 		OR
	(bCylinderRetractOutput	AND NOT  bCylinderRetractedInput) 	OR
	NOT ( bCylinderExtendedInput XOR bCylinderRetractedInput))	AND
	NOT bMoveNotAllowed THEN

		ton_Timeout.IN	:=	TRUE;
ELSE
		ton_Timeout.IN	:=	FALSE;
END_IF

ton_Timeout(IN:= , PT:= tTimeOut, Q=> bErrorPosition  , ET=> );

END_FUNCTION_BLOCK

// ---- POUs/METS/Common LIB/07_DEVICE LIB/Cylinders/FB_CylinderWithMeasur.TcPOU
FUNCTION_BLOCK FB_CylinderWithMeasur
VAR_INPUT

	bEnable				: BOOL;

	bPresureError			: BOOL;
	bSensorError			: BOOL;

	bCylinderExtendOutput	: BOOL;
	bCylinderRetractOutput	: BOOL;

	nTickInitNo		: UINT;
	nExtendTickLimit		: UINT := 65535;
	nExtendTickNo		: UINT := 64000;
	nRetractTcikNo		: UINT := 1000;
	nRetractTcikLimit		: UINT := 0;

END_VAR

VAR_OUTPUT

	bDeviceDisable		: BOOL;

	nTickNo		: UINT;
	bCylinderRetractedInput	: BOOL;
	bCylinderExtendedInput	: BOOL;

END_VAR
VAR
END_VAR

(********************************(Enable )**********************************************************)
IF NOT bEnable THEN

	bDeviceDisable :=	TRUE;

	nTickNo := nTickInitNo;
	bCylinderRetractedInput	:=	FALSE;
	bCylinderExtendedInput	:=	FALSE;

	RETURN;
ELSE

	bDeviceDisable :=	FALSE;
END_IF

(********************************(Operational Mode )**********************************************************)

	IF bCylinderExtendOutput  AND NOT bPresureError AND nTickNo <> nExtendTickLimit THEN
		nTickNo := LIMIT( nRetractTcikLimit, nTickNo + 1, nExtendTickLimit);
	END_IF

	IF bCylinderRetractOutput AND NOT bPresureError AND nTickNo <> nRetractTcikLimit THEN
		nTickNo := LIMIT( nRetractTcikLimit, nTickNo - 1, nExtendTickLimit);
	END_IF

	IF nTickNo <= nRetractTcikNo  AND NOT bSensorError THEN
		bCylinderRetractedInput:= TRUE;
	ELSE
		bCylinderRetractedInput := FALSE;
	END_IF

	IF nTickNo >= nExtendTickNo AND NOT bSensorError THEN
		bCylinderExtendedInput:= TRUE;
	ELSE
		bCylinderExtendedInput := FALSE;
	END_IF

END_FUNCTION_BLOCK

// ---- POUs/METS/Common LIB/07_DEVICE LIB/Door/FB_DOOR_RejectCtrl.TcPOU
FUNCTION_BLOCK FB_DOOR_RejectCtrl
VAR_INPUT
	bDoorOpenZone1			: BOOL;
	stDoorSettingsZone1			: ST_SYSTEM_Door;
	bDoorOpenZone2			: BOOL;
	stDoorSettingsZone2			: ST_SYSTEM_Door;
	stCTDateTime				: ST_SYSTEM_DateTime;
	sMetsDisplayCode			: T_MaxString;
END_VAR
VAR_OUTPUT
	stDoorOpenReject			: ST_SYSTEM_Door;
	bClearConveyorQueue	: BOOL;
	bClearPackerQueue		: BOOL;
	bClearCaseQueue		: BOOL;
END_VAR
VAR_IN_OUT
	stConveyorQueue						: ST_CASE_InfeedQueue;
	aPackerQueue							: ARRAY [0..1] OF ST_CASE_InfeedQueue;
	stCaseQueue							: ST_CASE_CaseQueue;
END_VAR
VAR
	stDoorOpenRejectZone1		: ST_SYSTEM_Door;
	stDoorOpenRejectZone2		: ST_SYSTEM_Door;
	nIndex: INT;
	nMaxCaseIndex		: INT;
END_VAR

bClearCaseQueue 		:= FALSE;
bClearConveyorQueue	:= FALSE;
bClearPackerQueue		:= FALSE;

nMaxCaseIndex := UDINT_TO_INT(SIZEOF(stCaseQueue.stCACData) / SIZEOF(stCaseQueue.stCACData[1]));

IF bDoorOpenZone1 THEN
	stDoorOpenRejectZone1:=stDoorSettingsZone1;
ELSE
	MEMSET(ADR(stDoorOpenRejectZone1), 16#00, SIZEOF(stDoorOpenRejectZone1));
END_IF

IF bDoorOpenZone2 THEN
	stDoorOpenRejectZone2:=stDoorSettingsZone2;
ELSE
	MEMSET(ADR(stDoorOpenRejectZone2), 16#00, SIZEOF(stDoorOpenRejectZone2));
END_IF

stDoorOpenReject.bClearConveyorQueue:=stDoorOpenRejectZone1.bClearConveyorQueue OR stDoorOpenRejectZone2.bClearConveyorQueue;
stDoorOpenReject.bClearPackerQueue:=stDoorOpenRejectZone1.bClearPackerQueue OR stDoorOpenRejectZone2.bClearPackerQueue;

FOR nIndex:=1 TO nMaxCaseIndex DO
	stDoorOpenReject.aClearCaseQueue[nIndex]:=stDoorOpenRejectZone1.aClearCaseQueue[nIndex] OR stDoorOpenRejectZone2.aClearCaseQueue[nIndex];
	IF stDoorOpenReject.aClearCaseQueue[nIndex] THEN
		bClearCaseQueue := TRUE;
	END_IF
END_FOR


bClearConveyorQueue	:= stDoorOpenReject.bClearConveyorQueue;
bClearPackerQueue		:= stDoorOpenReject.bClearPackerQueue;

IF stDoorOpenReject.bClearConveyorQueue THEN
	MEMSET(ADR(stConveyorQueue), 16#00, SIZEOF(stConveyorQueue));
	stConveyorQueue.bDoorReject := TRUE;
END_IF
IF stDoorOpenReject.bClearPackerQueue THEN
	MEMSET(ADR(aPackerQueue), 16#00, SIZEOF(aPackerQueue));
	aPackerQueue[0].bDoorReject := TRUE;
	aPackerQueue[1].bDoorReject := TRUE;
END_IF
FOR nIndex := 1 TO nMaxCaseIndex DO
	IF stDoorOpenReject.aClearCaseQueue[nIndex]  AND stCaseQueue.stCACData[nIndex].CodingAndTrackingMode > 0 THEN
		MEMSET(ADR(stCaseQueue.stCACData[nIndex]), 16#00, SIZEOF(stCaseQueue.stCACData[nIndex]));
		stCaseQueue.stCACData[nIndex].RejectCode := sMetsDisplayCode;
		stCaseQueue.stCACData[nIndex].ProductionDate := F_StringWildcard('#YYYYMMDD#', stCTDateTime.sSystemTime);
		stCaseQueue.stCACData[nIndex].ProductionTime := F_StringWildcard('#hhmmss#', stCTDateTime.sSystemTime);
		stCaseQueue.stCACData[nIndex].ProductionTimeOffset := F_SYSTEM_SystemTimeOffsetToHHMM(stCTDateTime.nSystemTimeOffset);
	END_IF
END_FOR

END_FUNCTION_BLOCK

// ---- POUs/METS/Common LIB/07_DEVICE LIB/Encoders/FB_ENCODER_AbsValueToPos.TcPOU
FUNCTION_BLOCK FB_ENCODER_AbsValueToPos
(* this block is used to calculate position from a row value of absolute encoder *)
VAR_INPUT
	i_nEncoderValue					:UDINT; (*current value from encoder (current increment)*)
	i_bInvertDirection		 		:BOOL;
	i_bResetPosition				:BOOL;
	i_nEncoderIncrements			:UDINT; (*Steps per revolution, encoder resolution*)
	i_fWheelDiameter_mm				:LREAL; (*wheel diameter in milimeters*)
END_VAR
VAR_OUTPUT
	o_fPosition_mm					:LREAL; (* position in milimeters *)
	o_bError						:BOOL;
	o_sError						:STRING;
END_VAR
VAR
	bBlockInitialized				:BOOL := FALSE;
	n								:INT;

	fWheelCircumference_mm			:LREAL;
	fDistancePerIncrement_mm		:LREAL;

	aEncoderValues					:ARRAY[0..9] OF UDINT; (* save old values for more direction of rotation analisys and overflow detection *)

	nDeltaInc						:DINT;

	bRotatingInPositiveDirection	:BOOL;
	bRotatingInNegativeDirection	:BOOL;

	bIndicationsPositiveDirections	:INT;
	bIndicationsNegativeDirections	:INT;

END_VAR

(*================================================================================================================================*)
(* INITIALIZE *)
(*================================================================================================================================*)
(* initialize block on the first call *)
IF bBlockInitialized = FALSE THEN

	(* Fill encoder values array with current encoder value *)
	FOR n := 0 TO 9 DO
		aEncoderValues[n] := i_nEncoderValue;
	END_FOR

	bBlockInitialized := TRUE;
END_IF

(* reset errors *)
o_bError := FALSE;
o_sError := '';

(* to avoid division by 0 *)
IF i_nEncoderIncrements = 0 THEN
	o_bError := TRUE;
	o_sError := 'i_nEncoderIncrements value can not be 0';
	RETURN;
END_IF

(* get the current encoder value to the encoder values array *)
MEMMOVE(ADR(aEncoderValues[1]), ADR(aEncoderValues[0]), SIZEOF(aEncoderValues) - SIZEOF(aEncoderValues[0]));
aEncoderValues[0] := i_nEncoderValue;



(*================================================================================================================================*)
(* RUN calculations *)
(*================================================================================================================================*)

fWheelCircumference_mm := i_fWheelDiameter_mm * 3.141592653589793238462643; (* Pi constant *)
fDistancePerIncrement_mm := fWheelCircumference_mm / i_nEncoderIncrements;

(* determine direction of rotation ----------------------------------------------------------------*)
(* we have to do this because of the overflow. eg. while running in positive directon, overflow will generate one indication in negative direction, so we are looking at this change through few cycles *)
bIndicationsPositiveDirections := 0;
bIndicationsNegativeDirections := 0;

FOR n := 0 TO 4 DO
	IF aEncoderValues[n] > aEncoderValues[n+1] THEN
		bIndicationsPositiveDirections := bIndicationsPositiveDirections + 1;

	ELSIF aEncoderValues[n] < aEncoderValues[n+1] THEN
		bIndicationsNegativeDirections := bIndicationsNegativeDirections + 1;

	END_IF
END_FOR;


bRotatingInPositiveDirection := FALSE;
bRotatingInNegativeDirection := FALSE;

IF bIndicationsPositiveDirections >= 3 AND bIndicationsPositiveDirections > bIndicationsNegativeDirections THEN
	bRotatingInPositiveDirection := TRUE;

ELSIF bIndicationsNegativeDirections >= 3 AND bIndicationsNegativeDirections > bIndicationsPositiveDirections THEN
	bRotatingInNegativeDirection := TRUE;

END_IF


(* calculate number of increments since last block call -----------------------------------------------------*)

(* positive overflow detected *)
IF 		bRotatingInPositiveDirection
	AND aEncoderValues[0] < aEncoderValues[1]
	AND ABS(UDINT_TO_REAL(aEncoderValues[0]) - UDINT_TO_REAL(aEncoderValues[1])) > UDINT_TO_REAL(i_nEncoderIncrements)/2 (* just to be sure difference has to be more then half circle. This helps with signal jitter issues *)
THEN
	nDeltaInc := 		REAL_TO_DINT((UDINT_TO_REAL(i_nEncoderIncrements) - UDINT_TO_REAL(aEncoderValues[1]))	(* from previous encoder value till the end of full rotation *)
					+	1 											(* from end of rotation to next turn *)
					+	UDINT_TO_REAL(aEncoderValues[0]));							(* from 0 till new encoder position *)

(* negative overflow detected *)
ELSIF 	bRotatingInNegativeDirection
	AND aEncoderValues[0] > aEncoderValues[1]
	AND ABS(UDINT_TO_REAL(aEncoderValues[0]) - UDINT_TO_REAL(aEncoderValues[1])) > UDINT_TO_REAL(i_nEncoderIncrements)/2 (* just to be sure difference has to be more then half circle. This helps with signal jitter issues *)
THEN

	nDeltaInc := 		REAL_TO_DINT((0 - UDINT_TO_REAL(aEncoderValues[1]))						(* from previous encoder value till the beginning of full rotation *)
					-	1 											(* from begginning of rotation to next turn *)
					-	(UDINT_TO_REAL(i_nEncoderIncrements) - UDINT_TO_REAL(aEncoderValues[0])));	(* from full turn value to new encoder position *)

(* expected scenario without overflow *)
ELSIF 	bRotatingInPositiveDirection AND aEncoderValues[0] > aEncoderValues[1]
	OR	bRotatingInNegativeDirection AND aEncoderValues[0] < aEncoderValues[1]
THEN
	nDeltaInc := REAL_TO_DINT(UDINT_TO_REAL(aEncoderValues[0]) - UDINT_TO_REAL(aEncoderValues[1]));

(* unexpected scenario. Can be caused by jitter in stationary position *)
ELSE
	nDeltaInc := 0;
END_IF




(* calculate current postiion ----------------------------------------------------------------*)
IF i_bResetPosition THEN
	o_fPosition_mm := 0;
ELSE
	IF i_bInvertDirection THEN
		o_fPosition_mm := o_fPosition_mm - nDeltaInc * fDistancePerIncrement_mm;
	ELSE
		o_fPosition_mm := o_fPosition_mm + nDeltaInc * fDistancePerIncrement_mm;
	END_IF
END_IF

END_FUNCTION_BLOCK

// ---- POUs/METS/Common LIB/07_DEVICE LIB/Encoders/FB_ENCODER_CamCtrl.TcPOU
FUNCTION_BLOCK FB_ENCODER_CamCtrl
VAR_INPUT
	bReadCams						: BOOL;
	bWriteCams						: BOOL;
	sAMSNetID						: T_AmsNetID;
	nSlaveAddr						: UINT;
	_fScalingFactor					: LREAL := 0.001373291015625; (* 360/262144 *)
END_VAR
VAR_OUTPUT
	bCam1							: BOOL;
	bCam2							: BOOL;
	bCam3							: BOOL;
	bCam4							: BOOL;
	bCam5							: BOOL;
	bCam6							: BOOL;
	bCam7							: BOOL;
	bCam8							: BOOL;
	fTemp							: LREAL;
	fActualValue					: LREAL;
END_VAR
VAR_IN_OUT
	stCamsHMi						: ARRAY[1..8] OF ST_AFS60_CamHMi;
	nZeroPosition					: UDINT;
	stAFS50CamStatus				: ST_AFS60_Status;
	(* IO *)
	nTemp							: UINT; (* AT%I*		: UINT;*)
	nCam1State						: USINT; (* AT%I*		: USINT; *)
	nPosValue						: UDINT; (* AT%I*		: UDINT; *)
	nMsecUpTime					: UDINT; (* AT%I*		: UDINT; *)
END_VAR
VAR


	_bCompleteAccess				: BOOL := TRUE;
	_ReadCams						: UINT;
	_WriteCams						: UINT;
	_CamNumber						: UINT;
	_TempEnabled					: UINT;
	_Hours							: UINT;
	_Minutes						: UINT;
	_Seconds						: UINT;
	_Time							: TIME;
	_nMSTemp						: UDINT;
	fbReadTrig						: R_TRIG;
	fbWriteTrig						: R_TRIG;
	fbEcCoESdoReadEx				: FB_EcCoESdoReadEx;
	fbEcCoESdoWriteEx				: FB_EcCoESdoWriteEx;
	_stCams							: ARRAY[1..8] OF ST_AFS60_Cam;
	bDebug: BOOL;
	fDebug1: LREAL;
	fDebug2: LREAL;
	fDebug3: LREAL;
	fDebug4: LREAL;
	fDebug5: LREAL;
	fDebug6: LREAL;
	fDebug7: LREAL;
	fDebug8: LREAL;
END_VAR

(* A bit crude *)
bCam1 := nCam1State.0;
bCam2 := nCam1State.1;
bCam3 := nCam1State.2;
bCam4 := nCam1State.3;
bCam5 := nCam1State.4;
bCam6 := nCam1State.5;
bCam7 := nCam1State.6;
bCam8 := nCam1State.7;

(* its the same thing *)
fTemp := nTemp;

(* A lot of faffing to get 2dp *)
fActualValue := UDINT_TO_LREAL(LREAL_TO_UDINT((UDINT_TO_LREAL(nPosValue) * _fScalingFactor) * 100)) / 100;

stAFS50CamStatus.bCam1 := bCam1;
stAFS50CamStatus.bCam2 := bCam2;
stAFS50CamStatus.bCam3 := bCam3;
stAFS50CamStatus.bCam4 := bCam4;
stAFS50CamStatus.bCam5 := bCam5;
stAFS50CamStatus.bCam6 := bCam6;
stAFS50CamStatus.bCam7 := bCam7;
stAFS50CamStatus.bCam8 := bCam8;

stAFS50CamStatus.fActualValue := fActualValue;
stAFS50CamStatus.fTemp := fTemp;
stAFS50CamStatus.nMsecUpTime := nMsecUpTime;


_Time := UDINT_TO_TIME(nMsecUpTime);
_Hours := UDINT_TO_UINT(nMsecUpTime / 1000 / 60 / 60);
_nMSTemp := nMsecUpTime - (_Hours * 1000 * 60 * 60);
_Minutes := UDINT_TO_UINT(_nMSTemp / 1000 / 60);
_nMSTemp := _nMSTemp - (_Minutes * 1000 * 60);
_Seconds := UDINT_TO_UINT(_nMSTemp / 1000 / 60);





(* READ CAMS *)
CASE _ReadCams OF

	0:
		fbReadTrig(CLK := bReadCams);
		IF fbReadTrig.Q THEN

			_CamNumber := 1;
			fbEcCoESdoReadEx(bExecute := FALSE);
			_ReadCams := _ReadCams + 1;

		END_IF
	(* ---------------------------------- *)

	1:
		(* Read Enabled *)
		fbEcCoESdoReadEx(
			sNetId:= sAMSNetID,
			nSlaveAddr:= nSlaveAddr,
			nSubIndex:= 1,
			nIndex:= 16#6302,
			pDstBuf:= ADR(_TempEnabled),
			cbBufLen:= 2,
			bExecute:= TRUE,
			tTimeout:= T#2.0S,
			bCompleteAccess:= _bCompleteAccess,
			bBusy=> ,
			bError=> ,
			nErrId=> );

		IF NOT fbEcCoESdoReadEx.bBusy THEN

			FOR _CamNumber := 1 TO 8 DO

				_stCams[_CamNumber].bEnable := GETBIT32(_TempEnabled, UINT_TO_BYTE(_CamNumber) - 1);

			END_FOR

			_CamNumber := 1;
			_ReadCams := _ReadCams + 1;
			fbEcCoESdoReadEx(bExecute := FALSE);


		END_IF
	(* ---------------------------------- *)

	2:
		(* Read Lower Limit *)
		fbEcCoESdoReadEx(
			sNetId:= sAMSNetID,
			nSlaveAddr:= nSlaveAddr,
			nSubIndex:= 1,
			nIndex:= 16#6310 + (_CamNumber - 1),
			pDstBuf:= ADR(_stCams[_CamNumber].nLowerLimit1),
			cbBufLen:= 8,
			bExecute:= TRUE,
			tTimeout:= T#2.0S,
			bCompleteAccess:= _bCompleteAccess,
			bBusy=> ,
			bError=> ,
			nErrId=> );

		IF NOT fbEcCoESdoReadEx.bBusy THEN

			_ReadCams := _ReadCams + 1;
			fbEcCoESdoReadEx(bExecute := FALSE);

		END_IF
	(* ---------------------------------- *)
	3:
		(* Read the Upper limit *)
		fbEcCoESdoReadEx(
			sNetId:= sAMSNetID,
			nSlaveAddr:= nSlaveAddr,
			nSubIndex:= 1,
			nIndex:= 16#6320 + (_CamNumber - 1),
			pDstBuf:= ADR(_stCams[_CamNumber].nUpperLimit1),
			cbBufLen:= 8,
			bExecute:= TRUE,
			tTimeout:= T#2.0S,
			bCompleteAccess:= _bCompleteAccess,
			bBusy=> ,
			bError=> ,
			nErrId=> );

		IF NOT fbEcCoESdoReadEx.bBusy THEN

			_CamNumber := _CamNumber + 1;

			IF _CamNumber > 8 THEN

				_ReadCams := _ReadCams + 1;

			ELSE

				_ReadCams := 2;
				fbEcCoESdoReadEx(bExecute := FALSE);

			END_IF

		END_IF
	(* ---------------------------------- *)

	4:
		FOR _CamNumber := 1 TO 8 DO

			stCamsHMi[_CamNumber].fLowerLimit1 := UDINT_TO_LREAL(_stCams[_CamNumber].nLowerLimit1) * _fScalingFactor;
			stCamsHMi[_CamNumber].fLowerLimit2 := UDINT_TO_LREAL(_stCams[_CamNumber].nLowerLimit2) * _fScalingFactor;
			stCamsHMi[_CamNumber].fUpperLimit1 := UDINT_TO_LREAL(_stCams[_CamNumber].nUpperLimit1) * _fScalingFactor;
			stCamsHMi[_CamNumber].fUpperLimit2 := UDINT_TO_LREAL(_stCams[_CamNumber].nUpperLimit2) * _fScalingFactor;
			stCamsHMi[_CamNumber].bEnable := _stCams[_CamNumber].bEnable;

		END_FOR

		_ReadCams := _ReadCams + 1;
	(* ---------------------------------- *)

	5 : (* Read Preset *)

		fbEcCoESdoReadEx(
			sNetId:= sAMSNetID,
			nSlaveAddr:= nSlaveAddr,
			nSubIndex:= 0,
			nIndex:= 16#6003,
			pDstBuf:= ADR(nZeroPosition),
			cbBufLen:= 8,
			bExecute:= TRUE,
			tTimeout:= T#2.0S,
			bCompleteAccess:= _bCompleteAccess,
			bBusy=> ,
			bError=> ,
			nErrId=> );

		IF NOT fbEcCoESdoReadEx.bBusy THEN

			fbEcCoESdoReadEx(bExecute := FALSE);

			_ReadCams := 0;
		END_IF

	(*-----------------------------------*)
END_CASE



(* WRITE CAMS *)
CASE _WriteCams OF

	0:
		fbWriteTrig(CLK := bWriteCams);
		IF fbWriteTrig.Q THEN

			bDebug := TRUE;
			FOR _CamNumber := 1 TO 8 DO

				_stCams[_CamNumber].bEnable := stCamsHMi[_CamNumber].bEnable;
				_stCams[_CamNumber].nLowerLimit1 := LREAL_TO_UDINT(F_SafeDIV(stCamsHMi[_CamNumber].fLowerLimit1, _fScalingFactor));
				_stCams[_CamNumber].nLowerLimit2 := LREAL_TO_UDINT(F_SafeDIV(stCamsHMi[_CamNumber].fLowerLimit2, _fScalingFactor));
				_stCams[_CamNumber].nUpperLimit1 := LREAL_TO_UDINT(F_SafeDIV(stCamsHMi[_CamNumber].fUpperLimit1, _fScalingFactor));
				_stCams[_CamNumber].nUpperLimit2 := LREAL_TO_UDINT(F_SafeDIV(stCamsHMi[_CamNumber].fUpperLimit2, _fScalingFactor));

			END_FOR

			fDebug1 := _stCams[7].nLowerLimit1 ;
			fDebug6 := stCamsHMi[7].fLowerLimit1 ;

			_CamNumber := 1;
			fbEcCoESdoWriteEx(bExecute := FALSE);
			_WriteCams := _WriteCams + 1;

		END_IF
	(* ---------------------------------- *)

	1:
		(* Write Enabled *)
		_TempEnabled := 0;
		FOR _CamNumber := 1 TO 8 DO

			IF _stCams[_CamNumber].bEnable THEN

			 _TempEnabled := DWORD_TO_UINT(SETBIT32(_TempEnabled, UINT_TO_BYTE(_CamNumber) - 1));

			END_IF

		END_FOR

		fbEcCoESdoWriteEx(
			sNetId:= sAMSNetID,
			nSlaveAddr:= nSlaveAddr,
			nSubIndex:= 1,
			nIndex:= 16#6302,
			pSrcBuf:= ADR(_TempEnabled),
			cbBufLen:= 2,
			bExecute:= TRUE,
			tTimeout:= T#2.0S,
			bCompleteAccess:= _bCompleteAccess,
			bBusy=> ,
			bError=> ,
			nErrId=> );

		IF NOT fbEcCoESdoWriteEx.bBusy THEN

			_CamNumber := 1;
			_WriteCams := _WriteCams + 1;
			fbEcCoESdoWriteEx(bExecute := FALSE);

			fDebug2 := _stCams[7].nLowerLimit1 ;
		END_IF
	(* ---------------------------------- *)

	2:
		(* Write Lower Limit *)
		fbEcCoESdoWriteEx(
			sNetId:= sAMSNetID,
			nSlaveAddr:= nSlaveAddr,
			nSubIndex:= 1,
			nIndex:= 16#6310 + (_CamNumber - 1),
			pSrcBuf:= ADR(_stCams[_CamNumber].nLowerLimit1),
			cbBufLen:= 8,
			bExecute:= TRUE,
			tTimeout:= T#2.0S,
			bCompleteAccess:= _bCompleteAccess,
			bBusy=> ,
			bError=> ,
			nErrId=> );

		IF NOT fbEcCoESdoWriteEx.bBusy THEN

			_WriteCams := _WriteCams + 1;
			fbEcCoESdoWriteEx(bExecute := FALSE);

			fDebug3 := _stCams[7].nLowerLimit1 ;

		END_IF
	(* ---------------------------------- *)
	3:
		(* Write the Upper limit *)
		fbEcCoESdoWriteEx(
			sNetId:= sAMSNetID,
			nSlaveAddr:= nSlaveAddr,
			nSubIndex:= 1,
			nIndex:= 16#6320 + (_CamNumber - 1),
			pSrcBuf:= ADR(_stCams[_CamNumber].nUpperLimit1),
			cbBufLen:= 8,
			bExecute:= TRUE,
			tTimeout:= T#2.0S,
			bCompleteAccess:= _bCompleteAccess,
			bBusy=> ,
			bError=> ,
			nErrId=> );

		IF NOT fbEcCoESdoWriteEx.bBusy THEN

			_CamNumber := _CamNumber + 1;

			IF _CamNumber > 8 THEN

				_WriteCams := _WriteCams + 1;
(*			_WriteCams := 0; (* debug *) *)
			fDebug4 := _stCams[7].nLowerLimit1 ;
			ELSE

				_WriteCams := 2;
				fbEcCoESdoWriteEx(bExecute := FALSE);

			END_IF

		END_IF
	(* ---------------------------------- *)

	4:  (* Write Preset *)

		fbEcCoESdoWriteEx(
			sNetId:= sAMSNetID,
			nSlaveAddr:= nSlaveAddr,
			nSubIndex:= 0,
			nIndex:= 16#6320 + (_CamNumber - 1),
			pSrcBuf:= ADR(nZeroPosition),
			cbBufLen:= 8,
			bExecute:= TRUE,
			tTimeout:= T#2.0S,
			bCompleteAccess:= _bCompleteAccess,
			bBusy=> ,
			bError=> ,
			nErrId=> );

		IF NOT fbEcCoESdoReadEx.bBusy THEN

			fDebug5 := _stCams[7].nLowerLimit1 ;

			fbEcCoESdoWriteEx(bExecute := FALSE);

			_WriteCams := 0;
		END_IF

	(*-----------------------------------*)

END_CASE

END_FUNCTION_BLOCK

// ---- POUs/METS/Common LIB/07_DEVICE LIB/Encoders/FB_ENCODER_SingleTurn.TcPOU
FUNCTION_BLOCK FB_ENCODER_SingleTurn
VAR_INPUT
	bStart				: BOOL;
	nEncoderPosition	: UDINT;
	bMotorUnitRun		: BOOL;
END_VAR
VAR_OUTPUT
	nOutputRevolutions: UDINT := 0;
	nOutputPulses: UDINT;
	nOutputMM: DINT;
END_VAR
VAR
	rtStartCounting: R_TRIG;
	rtSamplingCorrectionStart	: R_TRIG;
	rtSamplingCorrectionEnd	: R_TRIG;
	rtNewRevolution: R_TRIG;
	fScallingFactor: REAL := 1;
	nMaxEncoderValue:UDINT := 262144;
	fMaxDistanceValue:REAL := 160;
	nStartEncoderPosition: UDINT := 0;
	nPreviousEncoderPosition: UDINT := 0;
	bNewRevolution: BOOL;
	nPreviousOutputRevolutions  :UDINT;

	aLogEncoderSampling		: ARRAY[1..25] OF UDINT;
	nSamplingDiff				: UDINT;
	nPreviuseSamplingDiff		: UDINT;
	nOriginalStartPosition		: UDINT;
	nOriginalEndPosition		: UDINT;
	nSamplingCorrectionStart		: INT;
	nSamplingCorrectionEnd		: INT;
END_VAR

IF fScallingFactor = 1 THEN
	(* 1 mm -> 1638 encoder value*)
	fScallingFactor:=UDINT_TO_REAL(nMaxEncoderValue)/fMaxDistanceValue;
END_IF

rtStartCounting(CLK:=bStart);
IF rtStartCounting.Q THEN
	nOutputPulses:= 0;
	nOutputRevolutions:= 0;
	nPreviousOutputRevolutions:= 0;
	nStartEncoderPosition:=nEncoderPosition;
	nSamplingDiff:= 0;
END_IF
(*
MEMMOVE(ADR(aLogEncoderSampling[2]), ADR(aLogEncoderSampling[1]), SIZEOF(aLogEncoderSampling)-SIZEOF(aLogEncoderSampling[1]));
aLogEncoderSampling[1] := nEncoderPosition;

IF aLogEncoderSampling[2] <> 0 AND aLogEncoderSampling[3] <>0  THEN
	nSamplingDiff:= ABS(aLogEncoderSampling[2] - aLogEncoderSampling[3]);
END_IF
*)
rtSamplingCorrectionStart(CLK:=nSamplingDiff < nMaxEncoderValue/3 AND nSamplingDiff >10 AND  nStartEncoderPosition < LREAL_TO_UDINT(1.1*UDINT_TO_LREAL(nSamplingDiff))); (*3000*)(*2*nSamplingDiff*)
IF rtSamplingCorrectionStart.Q THEN

	nPreviuseSamplingDiff := nSamplingDiff;
	nOriginalStartPosition := nStartEncoderPosition;

	nSamplingCorrectionStart := nSamplingCorrectionStart + 1;

	nStartEncoderPosition := nMaxEncoderValue-LREAL_TO_UDINT(1.1*UDINT_TO_LREAL(nSamplingDiff)); (*2800*);(*(2*nSamplingDiff);*)
END_IF

rtSamplingCorrectionEnd(CLK:=nSamplingDiff < nMaxEncoderValue/3 AND nSamplingDiff >10 AND  nStartEncoderPosition > nMaxEncoderValue -LREAL_TO_UDINT(1.1*UDINT_TO_LREAL(nSamplingDiff))); (*3000*) (*3*nSamplingDiff*)
IF rtSamplingCorrectionEnd.Q THEN

	nPreviuseSamplingDiff := nSamplingDiff;
	nOriginalEndPosition := nStartEncoderPosition;

	nSamplingCorrectionEnd := nSamplingCorrectionEnd + 1;

	nStartEncoderPosition := nMaxEncoderValue- LREAL_TO_UDINT(1.15*UDINT_TO_LREAL(nSamplingDiff));(*3100**)(*(4*nSamplingDiff)*)
END_IF

rtNewRevolution(CLK:= bMotorUnitRun AND nStartEncoderPosition>nEncoderPosition);
IF rtNewRevolution.Q THEN
	nOutputRevolutions:= nOutputRevolutions + 1;
END_IF

IF bMotorUnitRun THEN

	MEMMOVE(ADR(aLogEncoderSampling[2]), ADR(aLogEncoderSampling[1]), SIZEOF(aLogEncoderSampling)-SIZEOF(aLogEncoderSampling[1]));
	aLogEncoderSampling[1] := nEncoderPosition;
	
	IF aLogEncoderSampling[2] <> 0 AND aLogEncoderSampling[3] <>0 AND ABS(aLogEncoderSampling[2] - aLogEncoderSampling[3]) < nMaxEncoderValue  THEN
		nSamplingDiff:= MAX(ABS(aLogEncoderSampling[2] - aLogEncoderSampling[3]), nSamplingDiff);
	END_IF

	IF nStartEncoderPosition<=nEncoderPosition THEN
		nOutputPulses:= nOutputRevolutions*nMaxEncoderValue + (nEncoderPosition - nStartEncoderPosition);
	ELSIF nOutputRevolutions> 0 THEN
		nOutputPulses:= (nOutputRevolutions-1)*nMaxEncoderValue + ((nMaxEncoderValue - nStartEncoderPosition) + nEncoderPosition);
	END_IF
END_IF
nPreviousOutputRevolutions:= nOutputRevolutions;
nPreviousEncoderPosition:=nEncoderPosition;


nOutputMM:= REAL_TO_DINT(UDINT_TO_REAL(nOutputPulses) / fScallingFactor);
(*nOutputMM:= nOutputPulses / fScallingFactor;*)

END_FUNCTION_BLOCK

// ---- POUs/METS/Common LIB/07_DEVICE LIB/IO2 Controls/FB_IO2_DoubleInputCtrl.TcPOU
FUNCTION_BLOCK FB_IO2_DoubleInputCtrl
VAR_INPUT
	eInputSource			: E_IO2_InputSource;

	bEnableInput1			: BOOL;
	eTypeInput1				: E_IO2_Type;
	tTimeOnFilter1			: TIME;
	tTimeOffFilter1			: TIME;

	bEnableInput2			: BOOL;
	eTypeInput2				: E_IO2_Type;
	tTimeOnFilter2			: TIME;
	tTimeOffFilter2			: TIME;
END_VAR
VAR_OUTPUT
	stProcessedInput		: ST_IO2_InputPLC;
END_VAR
VAR
	tTimeOnFilter			: TIME;
	tTimeOffFilter			: TIME;

	bInputState				: BOOL;
	rt_RawInput				: R_TRIG;
	ft_RawInput				: F_TRIG;

	ton_FilterONInput		: TON;
	tof_FilterOFFInput		: TOF;
	rt_ProcessedInput		: R_TRIG;
	ft_ProcessedInput		: F_TRIG;

END_VAR

CASE	eInputSource OF

E_IO2_InputSource.SENSOR:
	bInputState	:= SEL(eTypeInput1=E_IO2_Type.NO, NOT bEnableInput1, bEnableInput1);
	IF eTypeInput1 = E_IO2_Type.BLOCKED THEN bInputState := FALSE; END_IF

	tTimeOnFilter			:=	tTimeOnFilter1;
	tTimeOffFilter			:=	tTimeOffFilter1;
	
E_IO2_InputSource.MACHINE:
	bInputState	:= SEL(eTypeInput2=E_IO2_Type.NO, NOT bEnableInput2, bEnableInput2);
	IF eTypeInput2 = E_IO2_Type.BLOCKED THEN bInputState := FALSE; END_IF

	tTimeOnFilter			:=	tTimeOnFilter2;
	tTimeOffFilter			:=	tTimeOffFilter2;
ELSE
	bInputState	:= SEL(eTypeInput1=E_IO2_Type.NO, NOT bEnableInput1, bEnableInput1);
	IF eTypeInput1 = E_IO2_Type.BLOCKED THEN bInputState := FALSE; END_IF

	tTimeOnFilter			:=	tTimeOnFilter1;
	tTimeOffFilter			:=	tTimeOffFilter1;
END_CASE

stProcessedInput.bRawInput :=bInputState;
rt_RawInput(CLK:=stProcessedInput.bRawInput, Q=>stProcessedInput.bRawRTrigger);
ft_RawInput(CLK:=stProcessedInput.bRawInput, Q=>stProcessedInput.bRawFTrigger);

ton_FilterONInput(IN:=bInputState, PT:=tTimeOnFilter, Q=>);
IF ton_FilterONInput.Q THEN
	stProcessedInput.bStateInput := TRUE;
END_IF

tof_FilterOFFInput(IN:=bInputState, PT:=tTimeOffFilter, Q=>);
IF NOT tof_FilterOFFInput.Q THEN
	stProcessedInput.bStateInput := FALSE;
END_IF

rt_ProcessedInput(CLK:=stProcessedInput.bStateInput, Q=>stProcessedInput.bStateRTrigger);
ft_ProcessedInput(CLK:=stProcessedInput.bStateInput, Q=>stProcessedInput.bStateFTrigger);

END_FUNCTION_BLOCK

// ---- POUs/METS/Common LIB/07_DEVICE LIB/IO2 Controls/FB_IO2_DoubleInputLockCtrl.TcPOU
FUNCTION_BLOCK FB_IO2_DoubleInputLockCtrl
VAR_INPUT
	eInputSource		: E_IO2_InputSource;

	bEnableInput1		: BOOL;
	eTypeInput1			: E_IO2_Type;
	tTimeOnFilter1		: TIME;
	tTimeOffFilter1		: TIME;
	tTimeLatch1			: TIME;

	bEnableInput2		: BOOL;
	eTypeInput2			: E_IO2_Type;
	tTimeOnFilter2		: TIME;
	tTimeOffFilter2		: TIME;
	tTimeLatch2			: TIME;
END_VAR
VAR_OUTPUT
	stProcessedInput	: ST_IO2_InputPLC;
END_VAR
VAR
	tTimeOnFilter		: TIME;
	tTimeOffFilter		: TIME;

	bInputState			: BOOL;
	rt_RawInput			: R_TRIG;
	ft_RawInput			: F_TRIG;

	tTimeLatch			: TIME;
	tof_LockInput		: TOF;

	ton_FilterONInput	: TON;
	tof_FilterOFFInput	: TOF;
	rt_ProcessedInput	: R_TRIG;
	ft_ProcessedInput	: F_TRIG;

END_VAR

CASE	eInputSource OF

E_IO2_InputSource.SENSOR:
	bInputState	:= SEL(eTypeInput1=E_IO2_Type.NO, NOT bEnableInput1, bEnableInput1);
	IF eTypeInput1 = E_IO2_Type.BLOCKED THEN bInputState := FALSE; END_IF

	tTimeOnFilter			:=	tTimeOnFilter1;
	tTimeOffFilter			:=	tTimeOffFilter1;
	tTimeLatch			:=	tTimeLatch1;
	
E_IO2_InputSource.MACHINE:
	bInputState	:= SEL(eTypeInput2=E_IO2_Type.NO, NOT bEnableInput2, bEnableInput2);
	IF eTypeInput2 = E_IO2_Type.BLOCKED THEN bInputState := FALSE; END_IF

	tTimeOnFilter			:=	tTimeOnFilter2;
	tTimeOffFilter			:=	tTimeOffFilter2;
	tTimeLatch			:=	tTimeLatch2;
ELSE
	bInputState	:= SEL(eTypeInput1=E_IO2_Type.NO, NOT bEnableInput1, bEnableInput1);
	IF eTypeInput1 = E_IO2_Type.BLOCKED THEN bInputState := FALSE; END_IF

	tTimeOnFilter			:=	tTimeOnFilter1;
	tTimeOffFilter			:=	tTimeOffFilter1;
	tTimeLatch			:=	tTimeLatch1;
END_CASE

stProcessedInput.bRawInput :=bInputState;
rt_RawInput(CLK:=stProcessedInput.bRawInput, Q=>stProcessedInput.bRawRTrigger);
ft_RawInput(CLK:=stProcessedInput.bRawInput, Q=>stProcessedInput.bRawFTrigger);

tof_LockInput(IN:=bInputState, PT:=tTimeLatch, Q=>);

ton_FilterONInput(IN:=tof_LockInput.Q, PT:=tTimeOnFilter, Q=>);
IF ton_FilterONInput.Q THEN
	stProcessedInput.bStateInput := TRUE;
END_IF

tof_FilterOFFInput(IN:=tof_LockInput.Q, PT:=tTimeOffFilter, Q=>);
IF NOT tof_FilterOFFInput.Q THEN
	stProcessedInput.bStateInput := FALSE;
END_IF

rt_ProcessedInput(CLK:=stProcessedInput.bStateInput, Q=>stProcessedInput.bStateRTrigger);
ft_ProcessedInput(CLK:=stProcessedInput.bStateInput, Q=>stProcessedInput.bStateFTrigger);

END_FUNCTION_BLOCK

// ---- POUs/METS/Common LIB/07_DEVICE LIB/IO2 Controls/FB_IO2_ForceOutputs.TcPOU
FUNCTION_BLOCK FB_IO2_ForceOutputs
VAR_INPUT
	bEnable						: BOOL;
	sLabelName01					: STRING;
	sLabelName02					: STRING;
	sLabelName03					: STRING;
	sLabelName04					: STRING;
	sLabelName05					: STRING;
	sLabelName06					: STRING;
END_VAR
VAR_IN_OUT
	bForceOutput01				: BOOL;
	bForceOutput02				: BOOL;
	bForceOutput03				: BOOL;
	bForceOutput04				: BOOL;
	bForceOutput05				: BOOL;
	bForceOutput06				: BOOL;
END_VAR
VAR_OUTPUT
	aSetForceOutput				: ARRAY[1..6] OF ST_IO2_Diagnostic ;
	bOutputForceActive			: BOOL;
END_VAR

aSetForceOutput[1].sVarName		:= 	sLabelName01;
aSetForceOutput[2].sVarName		:= 	sLabelName02;
aSetForceOutput[3].sVarName		:= 	sLabelName03;
aSetForceOutput[4].sVarName		:= 	sLabelName04;
aSetForceOutput[5].sVarName		:= 	sLabelName05;
aSetForceOutput[6].sVarName		:= 	sLabelName06;

IF bEnable THEN
	aSetForceOutput[1].bState		:=	bForceOutput01;
	aSetForceOutput[1].sVarName		:= 	sLabelName01;
	aSetForceOutput[2].bState		:=	bForceOutput02;
	aSetForceOutput[2].sVarName		:= 	sLabelName02;
	aSetForceOutput[3].bState		:=	bForceOutput03;
	aSetForceOutput[3].sVarName		:= 	sLabelName03;
	aSetForceOutput[4].bState		:=	bForceOutput04;
	aSetForceOutput[4].sVarName		:= 	sLabelName04;
	aSetForceOutput[5].bState		:=	bForceOutput05;
	aSetForceOutput[5].sVarName		:= 	sLabelName05;
	aSetForceOutput[6].bState		:=	bForceOutput06;
	aSetForceOutput[6].sVarName		:= 	sLabelName06;
ELSE
	bForceOutput01				:= 	FALSE;
	bForceOutput02				:= 	FALSE;
	bForceOutput03				:= 	FALSE;
	bForceOutput04				:= 	FALSE;
	bForceOutput05				:= 	FALSE;
	bForceOutput06				:= 	FALSE;

	aSetForceOutput[1].bState		:=	bForceOutput01;
	aSetForceOutput[2].bState		:=	bForceOutput02;
	aSetForceOutput[3].bState		:=	bForceOutput03;
	aSetForceOutput[4].bState		:=	bForceOutput04;
	aSetForceOutput[5].bState		:=	bForceOutput05;
	aSetForceOutput[6].bState		:=	bForceOutput06;
END_IF

bOutputForceActive	:= bEnable;

END_FUNCTION_BLOCK

// ---- POUs/METS/Common LIB/07_DEVICE LIB/IO2 Controls/FB_IO2_OutputCtrl.TcPOU
FUNCTION_BLOCK FB_IO2_OutputCtrl
VAR_INPUT
	bEnable					: BOOL;
	eTypeOutput				: E_IO2_Type;
	tOutputDelayed			:TIME;
	tOutputLocked				:TIME;
END_VAR
VAR_OUTPUT
	bProcessedOutput						: BOOL;
	bProcessedDelayedOutput				: BOOL;
	bProcessedLockedOutput				: BOOL;
	bProcessedDelayedLockedOutput		: BOOL;
END_VAR
VAR
	tonDelayedOutputNO			: TON;
	tofLockedOutputNO			: TOF;
	tofDelayedLockedOutputNO	: TOF;

	tofDelayedOutputNC			: TOF;
	tonLockedOutputNC			: TON;
	tonDelayedLockedOutputNC	: TON;
END_VAR

bProcessedOutput:=SEL(eTypeOutput=E_IO2_Type.NO, NOT bEnable, bEnable);
IF eTypeOutput = E_IO2_Type.BLOCKED THEN bProcessedOutput := FALSE; END_IF

CASE eTypeOutput OF

E_IO2_Type.NO:
	tonDelayedOutputNO(IN:=bProcessedOutput, PT:=tOutputDelayed, Q=>bProcessedDelayedOutput);
	tofLockedOutputNO(IN:=bProcessedOutput, PT:=tOutputLocked, Q=>bProcessedLockedOutput);
	tofDelayedLockedOutputNO(IN:=bProcessedDelayedOutput, PT:=tOutputLocked, Q=>bProcessedDelayedLockedOutput);

E_IO2_Type.NC:
	tofDelayedOutputNC(IN:=bProcessedOutput, PT:=tOutputDelayed, Q=>bProcessedDelayedOutput);
	tonLockedOutputNC(IN:=bProcessedOutput, PT:=tOutputLocked, Q=>bProcessedLockedOutput);
	tonDelayedLockedOutputNC(IN:=bProcessedDelayedOutput, PT:=tOutputLocked, Q=>bProcessedDelayedLockedOutput);

ELSE

	bProcessedOutput						:= FALSE;
	bProcessedDelayedOutput				:= FALSE;
	bProcessedLockedOutput				:= FALSE;
	bProcessedDelayedLockedOutput		:= FALSE;
END_CASE
(*
bOutputState	:= SEL(eTypeInput=NO, NOT bEnable, bEnable);

tonDelayedOutput(IN:= bOutputState, PT:=tOutputDelayed, Q=>);
IF tonDelayedOutput.Q THEN
	bOutputProcessed := TRUE;
END_IF

tofLockedOutput(IN:=bOutputState, PT:=tOutputLocked, Q=>);
IF NOT tofLockedOutput.Q THEN
	bOutputProcessed := FALSE;
END_IF*)

END_FUNCTION_BLOCK

// ---- POUs/METS/Common LIB/07_DEVICE LIB/IO2 Controls/FB_IO2_SingleInputCtrl.TcPOU
FUNCTION_BLOCK FB_IO2_SingleInputCtrl
VAR_INPUT
	bEnable				: BOOL;
	eTypeInput 			: E_IO2_Type;
	tTimeOnFilter		: TIME;
	tTimeOffFilter 		: TIME;
END_VAR
VAR_OUTPUT
	stProcessedInput	: ST_IO2_InputPLC;
END_VAR
VAR
	bInputState			: BOOL;
	rt_RawInput			: R_TRIG;
	ft_RawInput			: F_TRIG;


	ton_FilterONInput	: TON;
	tof_FilterOFFInput	: TOF;
	rt_ProcessedInput	: R_TRIG;
	ft_ProcessedInput	: F_TRIG;

END_VAR

bInputState	:= SEL(eTypeInput=E_IO2_Type.NO, NOT bEnable, bEnable);
IF eTypeInput = E_IO2_Type.BLOCKED THEN bInputState := FALSE; END_IF

stProcessedInput.bRawInput :=bInputState;
rt_RawInput(CLK:=stProcessedInput.bRawInput, Q=>stProcessedInput.bRawRTrigger);
ft_RawInput(CLK:=stProcessedInput.bRawInput, Q=>stProcessedInput.bRawFTrigger);

ton_FilterONInput(IN:= bInputState, PT:=tTimeOnFilter, Q=>);
IF ton_FilterONInput.Q THEN
	stProcessedInput.bStateInput := TRUE;
END_IF

tof_FilterOFFInput(IN:=bInputState, PT:=tTimeOffFilter, Q=>);
IF NOT tof_FilterOFFInput.Q THEN
	stProcessedInput.bStateInput := FALSE;
END_IF

rt_ProcessedInput(CLK:=stProcessedInput.bStateInput, Q=>stProcessedInput.bStateRTrigger);
ft_ProcessedInput(CLK:=stProcessedInput.bStateInput, Q=>stProcessedInput.bStateFTrigger);

END_FUNCTION_BLOCK

// ---- POUs/METS/Common LIB/07_DEVICE LIB/IO2 Controls/FB_IO2_SingleInputLockCtrl.TcPOU
FUNCTION_BLOCK FB_IO2_SingleInputLockCtrl
VAR_INPUT
	bEnable				: BOOL;
	eTypeInput 			: E_IO2_Type;
	tTimeOnFilter		: TIME;
	tTimeOffFilter 		: TIME;
	tTimeLatch			: TIME;
END_VAR
VAR_OUTPUT
	stProcessedInput	: ST_IO2_InputPLC;
END_VAR
VAR
	bInputState			: BOOL;
	rt_RawInput			: R_TRIG;
	ft_RawInput			: F_TRIG;

	tof_LockInput		: TOF;

	ton_FilterONInput	: TON;
	tof_FilterOFFInput	: TOF;
	rt_ProcessedInput	: R_TRIG;
	ft_ProcessedInput	: F_TRIG;

END_VAR

bInputState	:= SEL(eTypeInput=E_IO2_Type.NO, NOT bEnable, bEnable);
IF eTypeInput = E_IO2_Type.BLOCKED THEN bInputState := FALSE; END_IF

stProcessedInput.bRawInput :=bInputState;
rt_RawInput(CLK:=stProcessedInput.bRawInput, Q=>stProcessedInput.bRawRTrigger);
ft_RawInput(CLK:=stProcessedInput.bRawInput, Q=>stProcessedInput.bRawFTrigger);

tof_LockInput(IN:=bInputState, PT:=tTimeLatch, Q=>);

ton_FilterONInput(IN:= tof_LockInput.Q, PT:=tTimeOnFilter, Q=>);
IF ton_FilterONInput.Q THEN
	stProcessedInput.bStateInput := TRUE;
END_IF

tof_FilterOFFInput(IN:=tof_LockInput.Q, PT:=tTimeOffFilter, Q=>);
IF NOT tof_FilterOFFInput.Q THEN
	stProcessedInput.bStateInput := FALSE;
END_IF

rt_ProcessedInput(CLK:=stProcessedInput.bStateInput, Q=>stProcessedInput.bStateRTrigger);
ft_ProcessedInput(CLK:=stProcessedInput.bStateInput, Q=>stProcessedInput.bStateFTrigger);

END_FUNCTION_BLOCK

// ---- POUs/METS/Common LIB/07_DEVICE LIB/IO2 Controls/FB_IO_ForceOutputs.TcPOU
FUNCTION_BLOCK FB_IO_ForceOutputs
VAR_INPUT
	bEnable							: BOOL;
END_VAR
VAR_IN_OUT
	bForceEUCAMachineRun_STCP		: BOOL;
	bForceCaseValidationOK_STCP		: BOOL;
	bForceOuterValidationOK_STCP	: BOOL;
	bForceLabellerInhibit_STL		: BOOL;
	bForceTPDMachineRun				: BOOL;
END_VAR
VAR_OUTPUT
	bSetEUCAMachineRun_STCP			: BOOL;	(*to set qb82KF1_1_EUCAMachineRun*)
	bSetCaseValidationOK_STCP		: BOOL;	(*to set qb82KF1_5_CaseValidationOK*)
	bSetOuterValidationOK_STCP		: BOOL;	(*to set qb82KF1_2_OuterValidationOK*)
	bSetLabellerInhibit_STL			: BOOL;	(*to set qb82KF1_3_LabellerInhibit_STL*)
	bSetTPDMachineRun				: BOOL;	(*to set qb482KF1_4_TPDMachineRun*)
END_VAR
VAR
END_VAR

IF bEnable THEN
	bSetEUCAMachineRun_STCP			:=	bForceEUCAMachineRun_STCP;
	bSetCaseValidationOK_STCP		:=	bForceCaseValidationOK_STCP;
	bSetOuterValidationOK_STCP		:=	bForceOuterValidationOK_STCP;
	bSetLabellerInhibit_STL			:=	bForceLabellerInhibit_STL;
	bSetTPDMachineRun				:=	bForceTPDMachineRun;
ELSE
	bForceEUCAMachineRun_STCP		:=	FALSE;
	bForceCaseValidationOK_STCP		:=	FALSE;
	bForceOuterValidationOK_STCP	:=	FALSE;
	bForceLabellerInhibit_STL		:=	FALSE;
	bForceTPDMachineRun				:=	FALSE;

	bSetEUCAMachineRun_STCP			:=	FALSE;
	bSetCaseValidationOK_STCP		:=	FALSE;
	bSetOuterValidationOK_STCP		:=	FALSE;
	bSetLabellerInhibit_STL			:=	FALSE;
	bSetTPDMachineRun				:=	FALSE;
END_IF

END_FUNCTION_BLOCK

// ---- POUs/METS/Common LIB/08_SOFTWARE LIB/AI Codes And Validation FBs/FB_CODE_ClearCodeInfo.TcPOU
FUNCTION_BLOCK FB_CODE_ClearCodeInfo
VAR_INPUT
END_VAR
VAR_IN_OUT
	stCodeInfo						: ST_CodeInfo;
END_VAR
VAR
	sMemoUserField					: STRING;
END_VAR

IF stCodeInfo.stGTIN.nListPosition = 0 THEN
	MEMSET(ADR(stCodeInfo.stGTIN), 16#00, SIZEOF(stCodeInfo.stGTIN));
	stCodeInfo.stGTIN.sFieldName :='GTIN';
	stCodeInfo.stGTIN.nGS1_AI := 1;
END_IF
IF stCodeInfo.stBatchID.nListPosition  = 0 THEN
	MEMSET(ADR(stCodeInfo.stBatchID), 16#00, SIZEOF(stCodeInfo.stBatchID));
	stCodeInfo.stBatchID.sFieldName :='BatchID';
	stCodeInfo.stBatchID.nGS1_AI := 10;
END_IF
IF stCodeInfo.stSerialCode.nListPosition = 0 THEN
	MEMSET(ADR(stCodeInfo.stSerialCode), 16#00, SIZEOF(stCodeInfo.stSerialCode));
	stCodeInfo.stSerialCode.sFieldName :='SerialCode';
	stCodeInfo.stSerialCode.nGS1_AI := 21;
END_IF
IF stCodeInfo.stProductionOrder.nListPosition  = 0 THEN
	MEMSET(ADR(stCodeInfo.stProductionOrder), 16#00, SIZEOF(stCodeInfo.stProductionOrder));
	stCodeInfo.stProductionOrder.sFieldName :='ProductionOrder';
	stCodeInfo.stProductionOrder.nGS1_AI := 91;
END_IF
IF stCodeInfo.stCryptoCode.nListPosition = 0 THEN
	MEMSET(ADR(stCodeInfo.stCryptoCode), 16#00, SIZEOF(stCodeInfo.stCryptoCode));
	stCodeInfo.stCryptoCode.sFieldName :='CryptoCode';
	stCodeInfo.stCryptoCode.nGS1_AI := 93;
END_IF
IF stCodeInfo.stRSKU.nListPosition = 0 THEN
	MEMSET(ADR(stCodeInfo.stRSKU), 16#00, SIZEOF(stCodeInfo.stRSKU));
	stCodeInfo.stRSKU.sFieldName :='SKU';
	stCodeInfo.stRSKU.nGS1_AI := 240;
END_IF
IF stCodeInfo.stMRP.nListPosition = 0 THEN
	MEMSET(ADR(stCodeInfo.stMRP), 16#00, SIZEOF(stCodeInfo.stMRP));
	stCodeInfo.stMRP.sFieldName :='MRP';
	stCodeInfo.stMRP.nGS1_AI := 8005;
END_IF
IF stCodeInfo.stBrandSpecification.nListPosition = 0 THEN
	MEMSET(ADR(stCodeInfo.stBrandSpecification), 16#00, SIZEOF(stCodeInfo.stBrandSpecification));
	stCodeInfo.stBrandSpecification.sFieldName := 'BrandSpec';
	stCodeInfo.stBrandSpecification.nGS1_AI := 92;
END_IF
IF stCodeInfo.stProduceDate.nListPosition = 0 THEN
	MEMSET(ADR(stCodeInfo.stProduceDate), 16#00, SIZEOF(stCodeInfo.stProduceDate));
	stCodeInfo.stProduceDate.sFieldName :='ProduceDate';
	stCodeInfo.stProduceDate.nGS1_AI := 94;
END_IF
IF stCodeInfo.stUserField3.nListPosition  = 0THEN
	sMemoUserField := stCodeInfo.stUserField3.sFieldName;
	MEMSET(ADR(stCodeInfo.stUserField3), 16#00, SIZEOF(stCodeInfo.stUserField3));
	stCodeInfo.stUserField3.sFieldName :=sMemoUserField;
	stCodeInfo.stUserField3.nGS1_AI := 95;
END_IF

END_FUNCTION_BLOCK

// ---- POUs/METS/Common LIB/08_SOFTWARE LIB/AI GS1 Codes And Validation FBs/FB_GS1_ClearCodeInfo.TcPOU
FUNCTION_BLOCK FB_GS1_ClearCodeInfo
VAR_INPUT
END_VAR
VAR_IN_OUT
	stCodeInfo						: ST_GS1_CodeInfo;
END_VAR
VAR
	nItemIndex		: INT ;
END_VAR

FOR nItemIndex :=1 TO cMAX_VALIDATION_ITEMS DO
	IF stCodeInfo.stGS1_Field[nItemIndex].eGS1_AIType = GS1_00   THEN
		MEMSET(ADR(stCodeInfo.stGS1_Field[nItemIndex]), 16#00, SIZEOF(stCodeInfo.stGS1_Field[nItemIndex]));
		stCodeInfo.stGS1_Field[nItemIndex].sFieldName :='Field Undefined';
	END_IF
END_FOR

END_FUNCTION_BLOCK

// ---- POUs/METS/Common LIB/08_SOFTWARE LIB/AI GS1 Codes And Validation FBs/FB_GS1_ValidateExplicitCode.TcPOU
 FUNCTION_BLOCK FB_GS1_ValidateExplicitCode
VAR_INPUT
	sFullCode					: T_MaxString;
	stCodeInfo				: ST_GS1_CodeInfo;
	stGS1_AI_Definition			: ST_GS1_AI_Definition;
END_VAR
VAR_OUTPUT
	bValidationOK				: BOOL;
	bEntireCodeLengthOK		: BOOL;

	(*bGS1_01_OK	: BOOL;
	bGS1_10_OK	: BOOL;
	bGS1_11_OK	: BOOL;
	bGS1_15_OK	: BOOL;
	bGS1_17_OK	: BOOL;
	bGS1_21_OK	: BOOL;
	bGS1_91_OK	: BOOL;
	bGS1_92_OK	: BOOL;
	bGS1_93_OK	: BOOL;
	bGS1_94_OK	: BOOL;
	bGS1_240_OK	: BOOL;
	bGS1_8005_OK	: BOOL;

	(*Fixed string lenght according to max string lenght form GS1*)
	sGS1_01		:STRING(14);
	sGS1_10		:STRING(20);
	sGS1_11		:STRING(6);
	sGS1_15		:STRING(6);
	sGS1_17		:STRING(6);
	sGS1_21		:STRING(21);
	sGS1_91		:STRING(90);
	sGS1_92		:STRING(90);
	sGS1_93		:STRING(90);
	sGS1_94		:STRING(90);
	sGS1_240		:STRING(30);
	sGS1_8005	:STRING(6);*)

END_VAR
VAR
	stItem			: ST_GS1_CodeValidation;
	nItemIndex		: INT;

	sAI_01ToValidateAgainst		: STRING(14);

	bGS1_01_OK	: BOOL;
	bGS1_10_OK	: BOOL;
	bGS1_11_OK	: BOOL;
	bGS1_15_OK	: BOOL;
	bGS1_17_OK	: BOOL;
	bGS1_21_OK	: BOOL;
	bGS1_240_OK	: BOOL;
	bGS1_8005_OK	: BOOL;
	bGS1_8006_OK	: BOOL;
	bGS1_8008_OK	: BOOL;
	bGS1_91_OK	: BOOL;
	bGS1_92_OK	: BOOL;
	bGS1_93_OK	: BOOL;
	bGS1_94_OK	: BOOL;

	bNON_GS1_01_OK	: BOOL;
	bNON_GS1_02_OK	: BOOL;
	bNON_GS1_03_OK	: BOOL;
	bNON_GS1_04_OK	: BOOL;
	bNON_GS1_05_OK	: BOOL;
	bNON_GS1_06_OK	: BOOL;
	bNON_GS1_07_OK	: BOOL;
	bNON_GS1_08_OK	: BOOL;
	bNON_GS1_09_OK	: BOOL;
	bNON_GS1_10_OK	: BOOL;

	(*Fixed string lenght according to max string lenght form GS1*)
	sGS1_01		:STRING(14);
	sGS1_10		:STRING(20);
	sGS1_11		:STRING(6);
	sGS1_15		:STRING(6);
	sGS1_17		:STRING(6);
	sGS1_21		:STRING(20);
	sGS1_240		:STRING(30);
	sGS1_8005	:STRING(6);
	sGS1_8006	:STRING(18);
	sGS1_8008	:STRING(12);
	sGS1_91		:STRING(90);
	sGS1_92		:STRING(90);
	sGS1_93		:STRING(90);
	sGS1_94		:STRING(90);

	sNON_GS1_01		:STRING(255);
	sNON_GS1_02		:STRING(255);
	sNON_GS1_03		:STRING(255);
	sNON_GS1_04		:STRING(255);
	sNON_GS1_05		:STRING(255);
	sNON_GS1_06		:STRING(255);
	sNON_GS1_07		:STRING(255);
	sNON_GS1_08		:STRING(255);
	sNON_GS1_09		:STRING(255);
	sNON_GS1_10		:STRING(255);

END_VAR

IF	stCodeInfo.nEntireLength = 0 THEN
	bEntireCodeLengthOK := FALSE;
	RETURN;
ELSIF	stCodeInfo.nEntireLength = stCodeInfo.nMinLength THEN
	bEntireCodeLengthOK := (LEN(sFullCode) = stCodeInfo.nEntireLength) OR NOT stCodeInfo.bValidateEntireLength;
ELSE
	bEntireCodeLengthOK := (LEN(sFullCode) >= stCodeInfo.nMinLength  AND   LEN(sFullCode) <= stCodeInfo.nEntireLength) OR NOT stCodeInfo.bValidateEntireLength;
END_IF

CASE stCodeInfo.eCodeLvlType OF

	E_LEVEL1:
		sAI_01ToValidateAgainst := stGS1_AI_Definition.stAI_01_Lvl1.sDataField;
	E_LEVEL2:
		sAI_01ToValidateAgainst := stGS1_AI_Definition.stAI_01_Lvl2.sDataField;
	E_LEVEL3:
		sAI_01ToValidateAgainst := stGS1_AI_Definition.stAI_01_Lvl3.sDataField;
ELSE
		sAI_01ToValidateAgainst := '';
END_CASE

sGS1_01		:='';
sGS1_10		:='';
sGS1_11		:='';
sGS1_15		:='';
sGS1_17		:='';
sGS1_21		:='';
sGS1_91		:='';
sGS1_92		:='';
sGS1_93		:='';
sGS1_94		:='';
sGS1_240		:='';
sGS1_8005	:='';

(*********************** GS1_01**************************************)
bGS1_01_OK := FALSE;
sGS1_01 := F_GS1_GetItem(sFullCode, GS1_01, stCodeInfo);

FOR nItemIndex :=1 TO cMAX_VALIDATION_ITEMS DO
	IF stCodeInfo.stGS1_Field[nItemIndex].eGS1_AIType =  GS1_01 THEN
		stItem := stCodeInfo.stGS1_Field[nItemIndex];
		IF stItem.bValidate THEN
			IF (LEN(sGS1_01) =  stItem.nCodeLength OR stItem.nCodeLength = 0)  AND  (sGS1_01 = sAI_01ToValidateAgainst OR sAI_01ToValidateAgainst = '') THEN
				bGS1_01_OK := TRUE;
			END_IF
		ELSE
			bGS1_01_OK := TRUE;
		END_IF
		EXIT;
	END_IF
END_FOR

(*********************** ********************************************)
(*********************** GS1_10**************************************)
bGS1_10_OK := FALSE;
sGS1_10 := F_GS1_GetItem(sFullCode, GS1_10, stCodeInfo);

FOR nItemIndex :=1 TO cMAX_VALIDATION_ITEMS DO
	IF stCodeInfo.stGS1_Field[nItemIndex].eGS1_AIType =  GS1_10 THEN
		stItem := stCodeInfo.stGS1_Field[nItemIndex];
		IF stItem.bValidate THEN
			IF (LEN(sGS1_10) = stItem.nCodeLength OR stItem.nCodeLength = 0) AND ( sGS1_10 =  stGS1_AI_Definition.stAI_10.sDataField OR stGS1_AI_Definition.stAI_10.sDataField = '') THEN
				bGS1_10_OK := TRUE;
			END_IF
		ELSE
			bGS1_10_OK := TRUE;
		END_IF
		EXIT;
	END_IF
END_FOR

(*********************** ********************************************)
(*********************** GS1_11**************************************)
bGS1_11_OK := FALSE;
sGS1_11 := F_GS1_GetItem(sFullCode, GS1_11, stCodeInfo);

FOR nItemIndex :=1 TO cMAX_VALIDATION_ITEMS DO
	IF stCodeInfo.stGS1_Field[nItemIndex].eGS1_AIType =  GS1_11 THEN
		stItem := stCodeInfo.stGS1_Field[nItemIndex];
		IF stItem.bValidate THEN
			IF (LEN(sGS1_11) = stItem.nCodeLength OR stItem.nCodeLength = 0)  AND  ( sGS1_11 =  stGS1_AI_Definition.stAI_11.sDataField OR stGS1_AI_Definition.stAI_11.sDataField = '')  THEN
				bGS1_11_OK := TRUE;
			END_IF
		ELSE
			bGS1_11_OK := TRUE;
		END_IF
		EXIT;
	END_IF
END_FOR

(*********************** ********************************************)
(*********************** GS1_15**************************************)
bGS1_15_OK := FALSE;
sGS1_15 := F_GS1_GetItem(sFullCode, GS1_15, stCodeInfo);

FOR nItemIndex :=1 TO cMAX_VALIDATION_ITEMS DO
	IF stCodeInfo.stGS1_Field[nItemIndex].eGS1_AIType =  GS1_15 THEN
		stItem := stCodeInfo.stGS1_Field[nItemIndex];
		IF stItem.bValidate THEN
			IF( LEN(sGS1_15) = stItem.nCodeLength OR stItem.nCodeLength = 0) AND  ( sGS1_15 =  stGS1_AI_Definition.stAI_15.sDataField OR stGS1_AI_Definition.stAI_15.sDataField = '')  THEN
				bGS1_15_OK := TRUE;
			END_IF
		ELSE
			bGS1_15_OK := TRUE;
		END_IF
		EXIT;
	END_IF
END_FOR

(*********************** ********************************************)
(*********************** GS1_17**************************************)
bGS1_17_OK := FALSE;
sGS1_17 := F_GS1_GetItem(sFullCode, GS1_17, stCodeInfo);

FOR nItemIndex :=1 TO cMAX_VALIDATION_ITEMS DO
	IF stCodeInfo.stGS1_Field[nItemIndex].eGS1_AIType =  GS1_17 THEN
		stItem := stCodeInfo.stGS1_Field[nItemIndex];
		IF stItem.bValidate THEN
			IF( LEN(sGS1_17) = stItem.nCodeLength OR stItem.nCodeLength = 0) AND  ( sGS1_17 =  stGS1_AI_Definition.stAI_17.sDataField OR stGS1_AI_Definition.stAI_17.sDataField = '')  THEN
				bGS1_17_OK := TRUE;
			END_IF
		ELSE
			bGS1_17_OK := TRUE;
		END_IF
		EXIT;
	END_IF
END_FOR

(*********************** ********************************************)
(*********************** GS1_21**************************************)
bGS1_21_OK := FALSE;
sGS1_21 := F_GS1_GetItem(sFullCode, GS1_21, stCodeInfo);

FOR nItemIndex :=1 TO cMAX_VALIDATION_ITEMS DO
	IF stCodeInfo.stGS1_Field[nItemIndex].eGS1_AIType =  GS1_21 THEN
		stItem := stCodeInfo.stGS1_Field[nItemIndex];
		IF stItem.bValidate THEN
			IF( LEN(sGS1_21) = stItem.nCodeLength OR stItem.nCodeLength = 0) AND  ( sGS1_21 =  stGS1_AI_Definition.stAI_21.sDataField OR stGS1_AI_Definition.stAI_21.sDataField = '')THEN
				bGS1_21_OK := TRUE;
			END_IF
		ELSE
			bGS1_21_OK := TRUE;
		END_IF
		EXIT;
	END_IF
END_FOR

(*********************** ********************************************)
(*********************** GS1_240**************************************)
bGS1_240_OK := FALSE;
sGS1_240 := F_GS1_GetItem(sFullCode, GS1_240, stCodeInfo);

FOR nItemIndex :=1 TO cMAX_VALIDATION_ITEMS DO
	IF stCodeInfo.stGS1_Field[nItemIndex].eGS1_AIType =  GS1_240 THEN
		stItem := stCodeInfo.stGS1_Field[nItemIndex];
		IF stItem.bValidate THEN
			IF (LEN(sGS1_240) = stItem.nCodeLength OR stItem.nCodeLength = 0) AND  ( sGS1_240 =  stGS1_AI_Definition.stAI_240.sDataField OR stGS1_AI_Definition.stAI_240.sDataField = '') THEN
				bGS1_240_OK := TRUE;
			END_IF
		ELSE
			bGS1_240_OK := TRUE;
		END_IF
		EXIT;
	END_IF
END_FOR

(*********************** ********************************************)
(*********************** GS1_8005************************************)
bGS1_8005_OK := FALSE;
sGS1_8005 := F_GS1_GetItem(sFullCode, GS1_8005, stCodeInfo);

FOR nItemIndex :=1 TO cMAX_VALIDATION_ITEMS DO
	IF stCodeInfo.stGS1_Field[nItemIndex].eGS1_AIType =  GS1_8005 THEN
		stItem := stCodeInfo.stGS1_Field[nItemIndex];
		IF stItem.bValidate THEN
			IF (LEN(sGS1_8005) = stItem.nCodeLength OR stItem.nCodeLength = 0) AND  ( sGS1_8005 =  stGS1_AI_Definition.stAI_8005.sDataField OR stGS1_AI_Definition.stAI_8005.sDataField = '') THEN
				bGS1_8005_OK := TRUE;
			END_IF
		ELSE
			bGS1_8005_OK := TRUE;
		END_IF
		EXIT;
	END_IF
END_FOR

(*********************** ********************************************)
(*********************** GS1_8006************************************)
bGS1_8006_OK := FALSE;
sGS1_8006 := F_GS1_GetItem(sFullCode, GS1_8006, stCodeInfo);

FOR nItemIndex :=1 TO cMAX_VALIDATION_ITEMS DO
	IF stCodeInfo.stGS1_Field[nItemIndex].eGS1_AIType =  GS1_8006 THEN
		stItem := stCodeInfo.stGS1_Field[nItemIndex];
		IF stItem.bValidate THEN
			IF (LEN(sGS1_8006) = stItem.nCodeLength OR stItem.nCodeLength = 0) AND  ( sGS1_8006 =  stGS1_AI_Definition.stAI_8006.sDataField OR stGS1_AI_Definition.stAI_8006.sDataField = '') THEN
				bGS1_8006_OK := TRUE;
			END_IF
		ELSE
			bGS1_8006_OK := TRUE;
		END_IF
		EXIT;
	END_IF
END_FOR

(*********************** ********************************************)
(*********************** GS1_8008************************************)
bGS1_8008_OK := FALSE;
sGS1_8008 := F_GS1_GetItem(sFullCode, GS1_8008, stCodeInfo);

FOR nItemIndex :=1 TO cMAX_VALIDATION_ITEMS DO
	IF stCodeInfo.stGS1_Field[nItemIndex].eGS1_AIType =  GS1_8008 THEN
		stItem := stCodeInfo.stGS1_Field[nItemIndex];
		IF stItem.bValidate THEN
			IF (LEN(sGS1_8008) = stItem.nCodeLength OR stItem.nCodeLength = 0) AND  ( sGS1_8008 =  stGS1_AI_Definition.stAI_8008.sDataField OR stGS1_AI_Definition.stAI_8008.sDataField = '') THEN
				bGS1_8008_OK := TRUE;
			END_IF
		ELSE
			bGS1_8008_OK := TRUE;
		END_IF
		EXIT;
	END_IF
END_FOR

(*********************** ********************************************)
(*********************** GS1_91**************************************)
bGS1_91_OK := FALSE;
sGS1_91 := F_GS1_GetItem(sFullCode, GS1_91, stCodeInfo);

FOR nItemIndex :=1 TO cMAX_VALIDATION_ITEMS DO
	IF stCodeInfo.stGS1_Field[nItemIndex].eGS1_AIType =  GS1_91 THEN
		stItem := stCodeInfo.stGS1_Field[nItemIndex];
		IF stItem.bValidate THEN
			IF (LEN(sGS1_91) = stItem.nCodeLength OR stItem.nCodeLength = 0)  AND  ( sGS1_91 =  stGS1_AI_Definition.stAI_91.sDataField OR stGS1_AI_Definition.stAI_91.sDataField = '') THEN
				bGS1_91_OK := TRUE;
			END_IF
		ELSE
			bGS1_91_OK := TRUE;
		END_IF
		EXIT;
	END_IF
END_FOR

(*********************** ********************************************)
(*********************** GS1_92**************************************)
bGS1_92_OK := FALSE;
sGS1_92 := F_GS1_GetItem(sFullCode, GS1_92, stCodeInfo);

FOR nItemIndex :=1 TO cMAX_VALIDATION_ITEMS DO
	IF stCodeInfo.stGS1_Field[nItemIndex].eGS1_AIType =  GS1_92 THEN
		stItem := stCodeInfo.stGS1_Field[nItemIndex];
		IF stItem.bValidate THEN
			IF (LEN(sGS1_92) = stItem.nCodeLength OR stItem.nCodeLength = 0) AND   ( sGS1_92 =  stGS1_AI_Definition.stAI_92.sDataField OR stGS1_AI_Definition.stAI_92.sDataField = '') THEN
				bGS1_92_OK := TRUE;
			END_IF
		ELSE
			bGS1_92_OK := TRUE;
		END_IF
		EXIT;
	END_IF
END_FOR

(*********************** ********************************************)
(*********************** GS1_93**************************************)
bGS1_93_OK := FALSE;
sGS1_93 := F_GS1_GetItem(sFullCode, GS1_93, stCodeInfo);

FOR nItemIndex :=1 TO cMAX_VALIDATION_ITEMS DO
	IF stCodeInfo.stGS1_Field[nItemIndex].eGS1_AIType =  GS1_93 THEN
		stItem := stCodeInfo.stGS1_Field[nItemIndex];
		IF stItem.bValidate THEN
			IF (LEN(sGS1_93) = stItem.nCodeLength OR stItem.nCodeLength = 0)  AND  ( sGS1_93 =  stGS1_AI_Definition.stAI_93.sDataField OR stGS1_AI_Definition.stAI_93.sDataField = '') THEN
				bGS1_93_OK := TRUE;
			END_IF
		ELSE
			bGS1_93_OK := TRUE;
		END_IF
		EXIT;
	END_IF
END_FOR

(*********************** ********************************************)
(*********************** GS1_94**************************************)
bGS1_94_OK := FALSE;
sGS1_94 := F_GS1_GetItem(sFullCode, GS1_94, stCodeInfo);

FOR nItemIndex :=1 TO cMAX_VALIDATION_ITEMS DO
	IF stCodeInfo.stGS1_Field[nItemIndex].eGS1_AIType =  GS1_94 THEN
		stItem := stCodeInfo.stGS1_Field[nItemIndex];
		IF stItem.bValidate THEN
			IF (LEN(sGS1_94) = stItem.nCodeLength OR stItem.nCodeLength = 0) AND  ( sGS1_94 =  stGS1_AI_Definition.stAI_94.sDataField OR stGS1_AI_Definition.stAI_94.sDataField = '') THEN
				bGS1_94_OK := TRUE;
			END_IF
		ELSE
			bGS1_94_OK := TRUE;
		END_IF
		EXIT;
	END_IF
END_FOR

(*********************** ********************************************)

(*********************** NON_GS1_01**************************************)
bNON_GS1_01_OK := FALSE;
sNON_GS1_01 := F_GS1_GetItem(sFullCode, NON_GS1_01, stCodeInfo);

FOR nItemIndex :=1 TO cMAX_VALIDATION_ITEMS DO
	IF stCodeInfo.stGS1_Field[nItemIndex].eGS1_AIType =  NON_GS1_01 THEN
		stItem := stCodeInfo.stGS1_Field[nItemIndex];
		IF stItem.bValidate THEN
			IF (LEN(sNON_GS1_01) = stItem.nCodeLength OR stItem.nCodeLength = 0) AND  ( sNON_GS1_01 =  stGS1_AI_Definition.stNON_GS1_01.sDataField OR stGS1_AI_Definition.stNON_GS1_01.sDataField = '') THEN
				bNON_GS1_01_OK := TRUE;
			END_IF
		ELSE
			bNON_GS1_01_OK := TRUE;
		END_IF
		EXIT;
	END_IF
END_FOR

(*********************** ********************************************)
(*********************** NON_GS1_02**************************************)
bNON_GS1_02_OK := FALSE;
sNON_GS1_02 := F_GS1_GetItem(sFullCode, NON_GS1_02, stCodeInfo);

FOR nItemIndex :=1 TO cMAX_VALIDATION_ITEMS DO
	IF stCodeInfo.stGS1_Field[nItemIndex].eGS1_AIType =  NON_GS1_02 THEN
		stItem := stCodeInfo.stGS1_Field[nItemIndex];
		IF stItem.bValidate THEN
			IF (LEN(sNON_GS1_02) = stItem.nCodeLength OR stItem.nCodeLength = 0) AND  ( sNON_GS1_02 =  stGS1_AI_Definition.stNON_GS1_02.sDataField OR stGS1_AI_Definition.stNON_GS1_02.sDataField = '') THEN
				bNON_GS1_02_OK := TRUE;
			END_IF
		ELSE
			bNON_GS1_02_OK := TRUE;
		END_IF
		EXIT;
	END_IF
END_FOR

(*********************** ********************************************)
(*********************** NON_GS1_03**************************************)
bNON_GS1_03_OK := FALSE;
sNON_GS1_03 := F_GS1_GetItem(sFullCode, NON_GS1_03, stCodeInfo);

FOR nItemIndex :=1 TO cMAX_VALIDATION_ITEMS DO
	IF stCodeInfo.stGS1_Field[nItemIndex].eGS1_AIType =  NON_GS1_03 THEN
		stItem := stCodeInfo.stGS1_Field[nItemIndex];
		IF stItem.bValidate THEN
			IF (LEN(sNON_GS1_03) = stItem.nCodeLength OR stItem.nCodeLength = 0) AND  ( sNON_GS1_03 =  stGS1_AI_Definition.stNON_GS1_03.sDataField OR stGS1_AI_Definition.stNON_GS1_03.sDataField = '') THEN
				bNON_GS1_03_OK := TRUE;
			END_IF
		ELSE
			bNON_GS1_03_OK := TRUE;
		END_IF
		EXIT;
	END_IF
END_FOR

(*********************** ********************************************)
(*********************** NON_GS1_04**************************************)
bNON_GS1_04_OK := FALSE;
sNON_GS1_04 := F_GS1_GetItem(sFullCode, NON_GS1_04, stCodeInfo);

FOR nItemIndex :=1 TO cMAX_VALIDATION_ITEMS DO
	IF stCodeInfo.stGS1_Field[nItemIndex].eGS1_AIType =  NON_GS1_04 THEN
		stItem := stCodeInfo.stGS1_Field[nItemIndex];
		IF stItem.bValidate THEN
			IF (LEN(sNON_GS1_04) = stItem.nCodeLength OR stItem.nCodeLength = 0) AND  ( sNON_GS1_04 =  stGS1_AI_Definition.stNON_GS1_04.sDataField OR stGS1_AI_Definition.stNON_GS1_04.sDataField = '') THEN
				bNON_GS1_04_OK := TRUE;
			END_IF
		ELSE
			bNON_GS1_04_OK := TRUE;
		END_IF
		EXIT;
	END_IF
END_FOR

(*********************** ********************************************)
(*********************** NON_GS1_05**************************************)
bNON_GS1_05_OK := FALSE;
sNON_GS1_05 := F_GS1_GetItem(sFullCode, NON_GS1_05, stCodeInfo);

FOR nItemIndex :=1 TO cMAX_VALIDATION_ITEMS DO
	IF stCodeInfo.stGS1_Field[nItemIndex].eGS1_AIType =  NON_GS1_05 THEN
		stItem := stCodeInfo.stGS1_Field[nItemIndex];
		IF stItem.bValidate THEN
			IF (LEN(sNON_GS1_05) = stItem.nCodeLength OR stItem.nCodeLength = 0) AND  ( sNON_GS1_05 =  stGS1_AI_Definition.stNON_GS1_05.sDataField OR stGS1_AI_Definition.stNON_GS1_05.sDataField = '') THEN
				bNON_GS1_05_OK := TRUE;
			END_IF
		ELSE
			bNON_GS1_05_OK := TRUE;
		END_IF
		EXIT;
	END_IF
END_FOR

(*********************** ********************************************)
(*********************** NON_GS1_06**************************************)
bNON_GS1_06_OK := FALSE;
sNON_GS1_06 := F_GS1_GetItem(sFullCode, NON_GS1_06, stCodeInfo);

FOR nItemIndex :=1 TO cMAX_VALIDATION_ITEMS DO
	IF stCodeInfo.stGS1_Field[nItemIndex].eGS1_AIType =  NON_GS1_06 THEN
		stItem := stCodeInfo.stGS1_Field[nItemIndex];
		IF stItem.bValidate THEN
			IF (LEN(sNON_GS1_06) = stItem.nCodeLength OR stItem.nCodeLength = 0) AND  ( sNON_GS1_06 =  stGS1_AI_Definition.stNON_GS1_06.sDataField OR stGS1_AI_Definition.stNON_GS1_06.sDataField = '') THEN
				bNON_GS1_06_OK := TRUE;
			END_IF
		ELSE
			bNON_GS1_06_OK := TRUE;
		END_IF
		EXIT;
	END_IF
END_FOR

(*********************** ********************************************)
(*********************** NON_GS1_07**************************************)
bNON_GS1_07_OK := FALSE;
sNON_GS1_07 := F_GS1_GetItem(sFullCode, NON_GS1_07, stCodeInfo);

FOR nItemIndex :=1 TO cMAX_VALIDATION_ITEMS DO
	IF stCodeInfo.stGS1_Field[nItemIndex].eGS1_AIType =  NON_GS1_07 THEN
		stItem := stCodeInfo.stGS1_Field[nItemIndex];
		IF stItem.bValidate THEN
			IF (LEN(sNON_GS1_07) = stItem.nCodeLength OR stItem.nCodeLength = 0) AND  ( sNON_GS1_07 =  stGS1_AI_Definition.stNON_GS1_07.sDataField OR stGS1_AI_Definition.stNON_GS1_07.sDataField = '') THEN
				bNON_GS1_07_OK := TRUE;
			END_IF
		ELSE
			bNON_GS1_07_OK := TRUE;
		END_IF
		EXIT;
	END_IF
END_FOR

(*********************** ********************************************)
(*********************** NON_GS1_08**************************************)
bNON_GS1_08_OK := FALSE;
sNON_GS1_08 := F_GS1_GetItem(sFullCode, NON_GS1_08, stCodeInfo);

FOR nItemIndex :=1 TO cMAX_VALIDATION_ITEMS DO
	IF stCodeInfo.stGS1_Field[nItemIndex].eGS1_AIType =  NON_GS1_08 THEN
		stItem := stCodeInfo.stGS1_Field[nItemIndex];
		IF stItem.bValidate THEN
			IF (LEN(sNON_GS1_08) = stItem.nCodeLength OR stItem.nCodeLength = 0) AND  ( sNON_GS1_08 =  stGS1_AI_Definition.stNON_GS1_08.sDataField OR stGS1_AI_Definition.stNON_GS1_08.sDataField = '') THEN
				bNON_GS1_08_OK := TRUE;
			END_IF
		ELSE
			bNON_GS1_08_OK := TRUE;
		END_IF
		EXIT;
	END_IF
END_FOR

(*********************** ********************************************)
(*********************** NON_GS1_09**************************************)
bNON_GS1_09_OK := FALSE;
sNON_GS1_09 := F_GS1_GetItem(sFullCode, NON_GS1_09, stCodeInfo);

FOR nItemIndex :=1 TO cMAX_VALIDATION_ITEMS DO
	IF stCodeInfo.stGS1_Field[nItemIndex].eGS1_AIType =  NON_GS1_09 THEN
		stItem := stCodeInfo.stGS1_Field[nItemIndex];
		IF stItem.bValidate THEN
			IF (LEN(sNON_GS1_09) = stItem.nCodeLength OR stItem.nCodeLength = 0) AND  ( sNON_GS1_09 =  stGS1_AI_Definition.stNON_GS1_09.sDataField OR stGS1_AI_Definition.stNON_GS1_09.sDataField = '') THEN
				bNON_GS1_09_OK := TRUE;
			END_IF
		ELSE
			bNON_GS1_09_OK := TRUE;
		END_IF
		EXIT;
	END_IF
END_FOR

(*********************** ********************************************)
(*********************** NON_GS1_10**************************************)
bNON_GS1_10_OK := FALSE;
sNON_GS1_10 := F_GS1_GetItem(sFullCode, NON_GS1_10, stCodeInfo);

FOR nItemIndex :=1 TO cMAX_VALIDATION_ITEMS DO
	IF stCodeInfo.stGS1_Field[nItemIndex].eGS1_AIType =  NON_GS1_10 THEN
		stItem := stCodeInfo.stGS1_Field[nItemIndex];
		IF stItem.bValidate THEN
			IF (LEN(sNON_GS1_10) = stItem.nCodeLength OR stItem.nCodeLength = 0) AND  ( sNON_GS1_10 =  stGS1_AI_Definition.stNON_GS1_10.sDataField OR stGS1_AI_Definition.stNON_GS1_10.sDataField = '') THEN
				bNON_GS1_10_OK := TRUE;
			END_IF
		ELSE
			bNON_GS1_10_OK := TRUE;
		END_IF
		EXIT;
	END_IF
END_FOR

(*********************** ********************************************)


bValidationOK	:= bEntireCodeLengthOK;

FOR nItemIndex :=1 TO cMAX_VALIDATION_ITEMS DO
	CASE stCodeInfo.stGS1_Field[nItemIndex].eGS1_AIType OF
	GS1_01:
		bValidationOK := bValidationOK AND bGS1_01_OK;
	GS1_10:
		bValidationOK := bValidationOK AND bGS1_10_OK;
	GS1_11:
		bValidationOK := bValidationOK AND bGS1_11_OK;
	GS1_15:
		bValidationOK := bValidationOK AND bGS1_15_OK;
	GS1_17:
		bValidationOK := bValidationOK AND bGS1_17_OK;
	GS1_21:
		bValidationOK := bValidationOK AND bGS1_21_OK;
	GS1_240:
		bValidationOK := bValidationOK AND bGS1_240_OK;
	GS1_8005:
		bValidationOK := bValidationOK AND bGS1_8005_OK;
	GS1_8006:
		bValidationOK := bValidationOK AND bGS1_8006_OK;
	GS1_8008:
		bValidationOK := bValidationOK AND bGS1_8008_OK;
	GS1_91:
		bValidationOK := bValidationOK AND bGS1_91_OK;
	GS1_92:
		bValidationOK := bValidationOK AND bGS1_92_OK;
	GS1_93:
		bValidationOK := bValidationOK AND bGS1_93_OK;
	GS1_94:
		bValidationOK := bValidationOK AND bGS1_94_OK;
	NON_GS1_01:
		bValidationOK := bValidationOK AND bNON_GS1_01_OK;
	NON_GS1_02:
		bValidationOK := bValidationOK AND bNON_GS1_02_OK;
	NON_GS1_03:
		bValidationOK := bValidationOK AND bNON_GS1_03_OK;
	NON_GS1_04:
		bValidationOK := bValidationOK AND bNON_GS1_04_OK;
	NON_GS1_05:
		bValidationOK := bValidationOK AND bNON_GS1_05_OK;
	NON_GS1_06:
		bValidationOK := bValidationOK AND bNON_GS1_06_OK;
	NON_GS1_07:
		bValidationOK := bValidationOK AND bNON_GS1_07_OK;
	NON_GS1_08:
		bValidationOK := bValidationOK AND bNON_GS1_08_OK;
	NON_GS1_09:
		bValidationOK := bValidationOK AND bNON_GS1_09_OK;
	NON_GS1_10:
		bValidationOK := bValidationOK AND bNON_GS1_10_OK;
	END_CASE
END_FOR

END_FUNCTION_BLOCK

// ---- POUs/METS/Common LIB/08_SOFTWARE LIB/AI GS1 Codes And Validation FBs/F_GS1_GetItem.TcPOU
FUNCTION F_GS1_GetItem : T_MaxString
VAR_INPUT
	sFullCode			: T_MaxString;
	eCodeAIType		: E_GS1_CodeAIType;
	stCodeInfo		: ST_GS1_CodeInfo;
END_VAR
VAR
	stItem			: ST_GS1_CodeValidation;
	nItemIndex		: INT;
	(*eCodeAIPattern	: E_CodeAIType;*)
	sItem			: T_MaxString;
	nStart			: INT;
	nEnd				: INT;
	sTemp			: T_MaxString;
END_VAR

IF stCodeInfo.nEntireLength > 0 THEN

